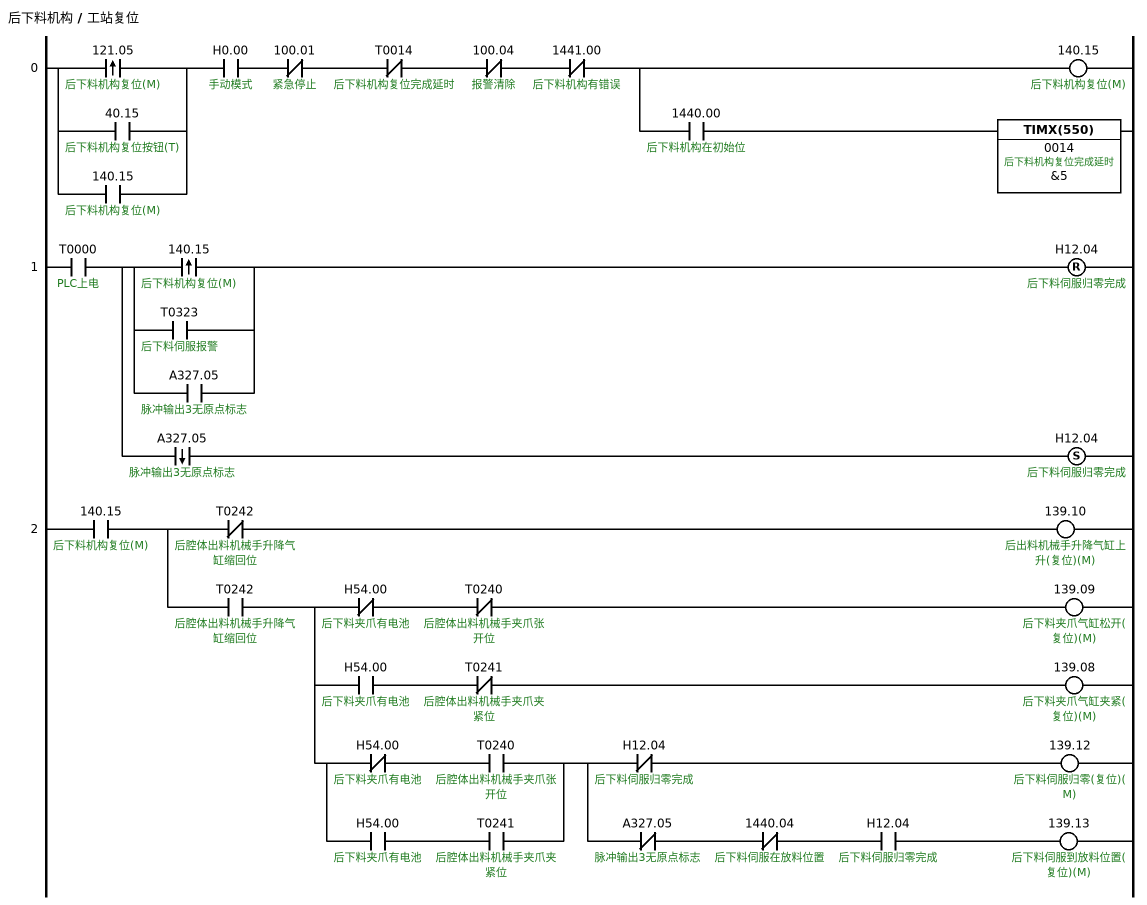
; [picture p216: 后下料机构 / 工站复位, rungs 0-2]
; rung 0
@LD 121.05  ; 后下料机构复位(M)
OR 40.15  ; 后下料机构复位按钮(T)
OR 140.15  ; 后下料机构复位(M)
AND H0.00  ; 手动模式
ANDNOT 100.01  ; 紧急停止
ANDNOT T0014  ; 后下料机构复位完成延时
ANDNOT 100.04  ; 报警清除
ANDNOT 1441.00  ; 后下料机构有错误
OUT 140.15  ; 后下料机构复位(M)
AND 1440.00  ; 后下料机构在初始位
TIMX(550) 0014 &5  ; 后下料机构复位完成延时
; rung 1
LD T0000  ; PLC上电
OUT TR0
@LD 140.15  ; 后下料机构复位(M)
OR T0323  ; 后下料伺服报警
OR A327.05  ; 脉冲输出3无原点标志
ANDLD
RSET H12.04  ; 后下料伺服归零完成
LD TR0
%AND A327.05  ; 脉冲输出3无原点标志
SET H12.04  ; 后下料伺服归零完成
; rung 2
LD 140.15  ; 后下料机构复位(M)
OUT TR0
ANDNOT T0242  ; 后腔体出料机械手升降气缸缩回位
OUT 139.10  ; 后出料机械手升降气缸上升(复位)(M)
LD TR0
AND T0242  ; 后腔体出料机械手升降气缸缩回位
OUT TR0
ANDNOT H54.00  ; 后下料夹爪有电池
ANDNOT T0240  ; 后腔体出料机械手夹爪张开位
OUT 139.09  ; 后下料夹爪气缸松开(复位)(M)
LD TR0
AND H54.00  ; 后下料夹爪有电池
ANDNOT T0241  ; 后腔体出料机械手夹爪夹紧位
OUT 139.08  ; 后下料夹爪气缸夹紧(复位)(M)
LD TR0
LDNOT H54.00  ; 后下料夹爪有电池
AND T0240  ; 后腔体出料机械手夹爪张开位
LD H54.00  ; 后下料夹爪有电池
AND T0241  ; 后腔体出料机械手夹爪夹紧位
ORLD
ANDLD
OUT TR0
ANDNOT H12.04  ; 后下料伺服归零完成
OUT 139.12  ; 后下料伺服归零(复位)(M)
LD TR0
ANDNOT A327.05  ; 脉冲输出3无原点标志
ANDNOT 1440.04  ; 后下料伺服在放料位置
AND H12.04  ; 后下料伺服归零完成
OUT 139.13  ; 后下料伺服到放料位置(复位)(M)

### Section 手动操作

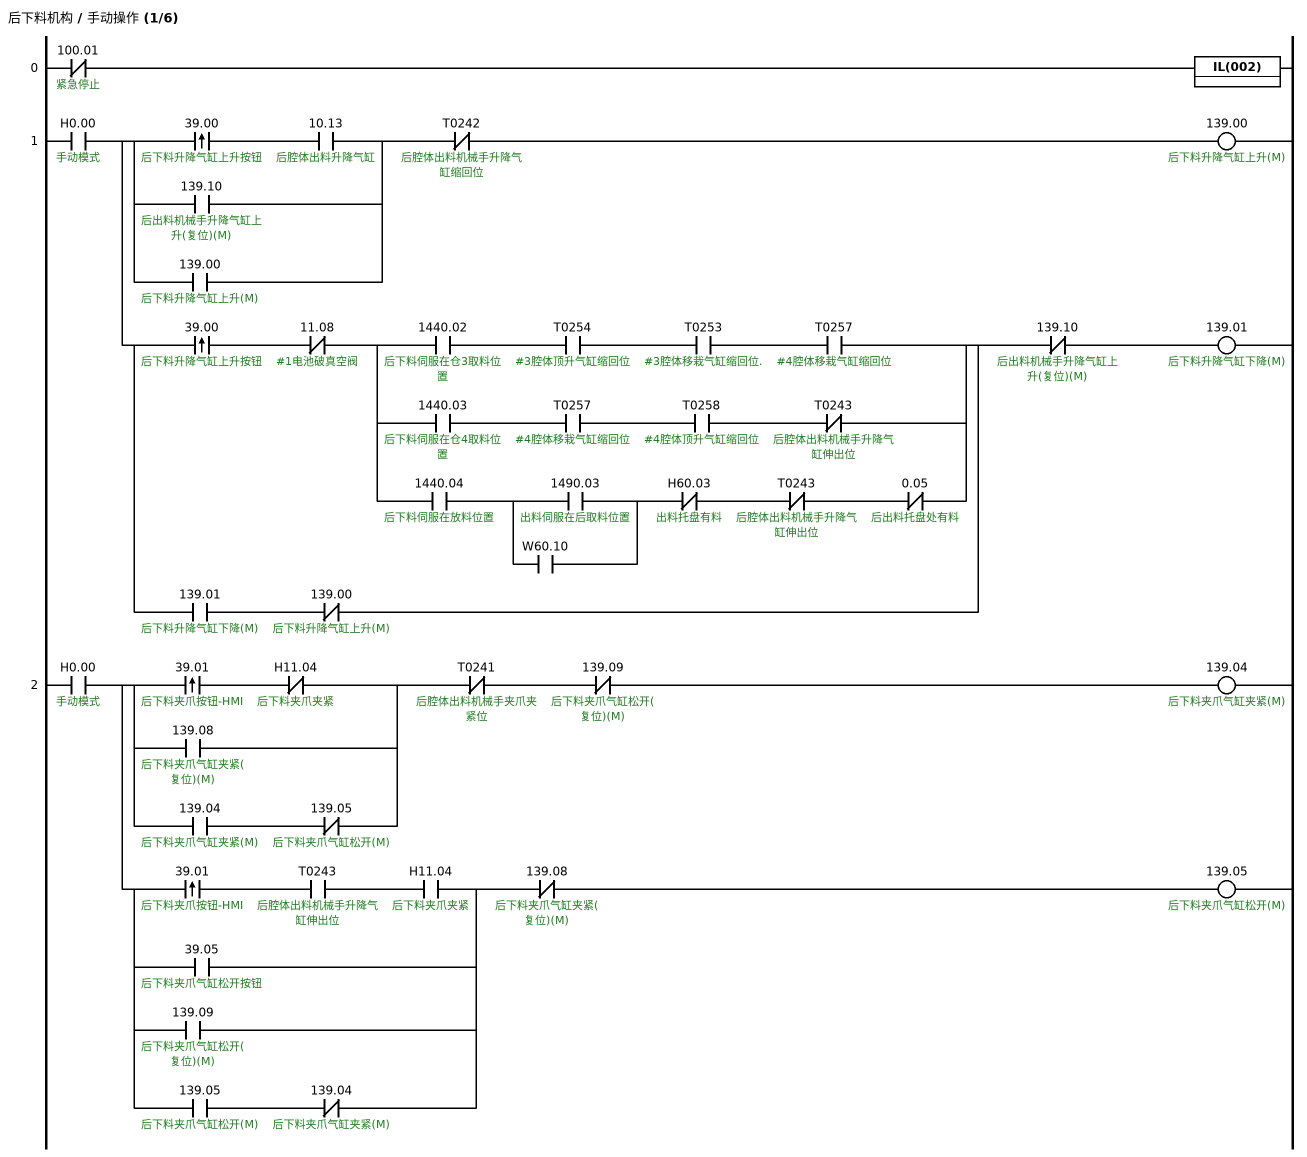
; rung 0
LDNOT 100.01  ; 紧急停止
IL(002)
; rung 1
LD H0.00  ; 手动模式
OUT TR0
@LD 39.00  ; 后下料升降气缸上升按钮
AND 10.13  ; 后腔体出料升降气缸
OR 139.10  ; 后出料机械手升降气缸上升(复位)(M)
OR 139.00  ; 后下料升降气缸上升(M)
ANDLD
ANDNOT T0242  ; 后腔体出料机械手升降气缸缩回位
OUT 139.00  ; 后下料升降气缸上升(M)
LD TR0
@LD 39.00  ; 后下料升降气缸上升按钮
ANDNOT 11.08  ; #1电池破真空阀
LD 1440.02  ; 后下料伺服在仓3取料位置
AND T0254  ; #3腔体顶升气缸缩回位
AND T0253  ; #3腔体移栽气缸缩回位.
AND T0257  ; #4腔体移栽气缸缩回位
LD 1440.03  ; 后下料伺服在仓4取料位置
AND T0257  ; #4腔体移栽气缸缩回位
AND T0258  ; #4腔体顶升气缸缩回位
ANDNOT T0243  ; 后腔体出料机械手升降气缸伸出位
ORLD
LD 1440.04  ; 后下料伺服在放料位置
LD 1490.03  ; 出料伺服在后取料位置
OR W60.10
ANDLD
ANDNOT H60.03  ; 出料托盘有料
ANDNOT T0243  ; 后腔体出料机械手升降气缸伸出位
ANDNOT 0.05  ; 后出料托盘处有料
ORLD
ANDLD
LD 139.01  ; 后下料升降气缸下降(M)
ANDNOT 139.00  ; 后下料升降气缸上升(M)
ORLD
ANDLD
ANDNOT 139.10  ; 后出料机械手升降气缸上升(复位)(M)
OUT 139.01  ; 后下料升降气缸下降(M)
; rung 2
LD H0.00  ; 手动模式
OUT TR0
@LD 39.01  ; 后下料夹爪按钮-HMI
ANDNOT H11.04  ; 后下料夹爪夹紧
OR 139.08  ; 后下料夹爪气缸夹紧(复位)(M)
LD 139.04  ; 后下料夹爪气缸夹紧(M)
ANDNOT 139.05  ; 后下料夹爪气缸松开(M)
ORLD
ANDLD
ANDNOT T0241  ; 后腔体出料机械手夹爪夹紧位
ANDNOT 139.09  ; 后下料夹爪气缸松开(复位)(M)
OUT 139.04  ; 后下料夹爪气缸夹紧(M)
LD TR0
@LD 39.01  ; 后下料夹爪按钮-HMI
AND T0243  ; 后腔体出料机械手升降气缸伸出位
AND H11.04  ; 后下料夹爪夹紧
OR 39.05  ; 后下料夹爪气缸松开按钮
OR 139.09  ; 后下料夹爪气缸松开(复位)(M)
LD 139.05  ; 后下料夹爪气缸松开(M)
ANDNOT 139.04  ; 后下料夹爪气缸夹紧(M)
ORLD
ANDLD
ANDNOT 139.08  ; 后下料夹爪气缸夹紧(复位)(M)
OUT 139.05  ; 后下料夹爪气缸松开(M)

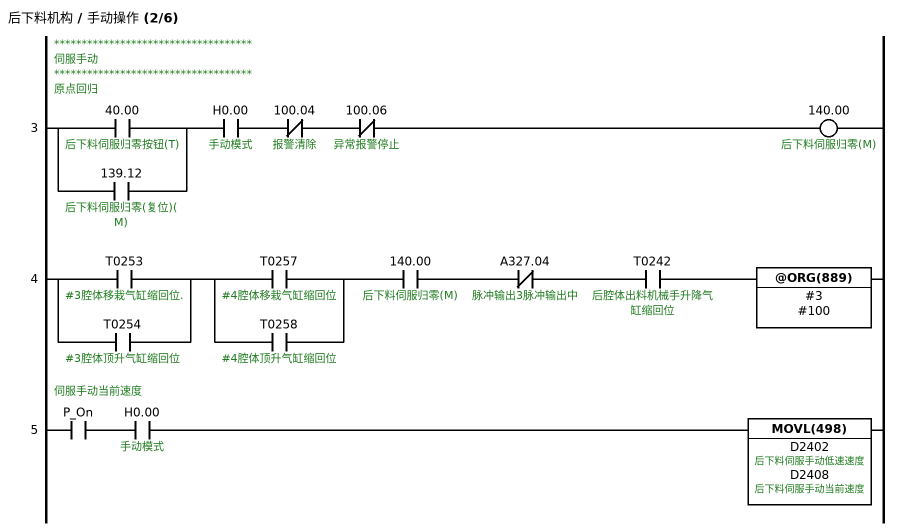
; rung 3: ************************************ / 伺服手动 / ************************************ / 原点回归
LD 40.00  ; 后下料伺服归零按钮(T)
OR 139.12  ; 后下料伺服归零(复位)(M)
AND H0.00  ; 手动模式
ANDNOT 100.04  ; 报警清除
ANDNOT 100.06  ; 异常报警停止
OUT 140.00  ; 后下料伺服归零(M)
; rung 4
LD T0253  ; #3腔体移栽气缸缩回位.
OR T0254  ; #3腔体顶升气缸缩回位
LD T0257  ; #4腔体移栽气缸缩回位
OR T0258  ; #4腔体顶升气缸缩回位
ANDLD
AND 140.00  ; 后下料伺服归零(M)
ANDNOT A327.04  ; 脉冲输出3脉冲输出中
AND T0242  ; 后腔体出料机械手升降气缸缩回位
@ORG(889) #3 #100
; rung 5: 伺服手动当前速度
LD P_On
AND H0.00  ; 手动模式
MOVL(498) D2402 D2408  ; 后下料伺服手动低速速度, 后下料伺服手动当前速度

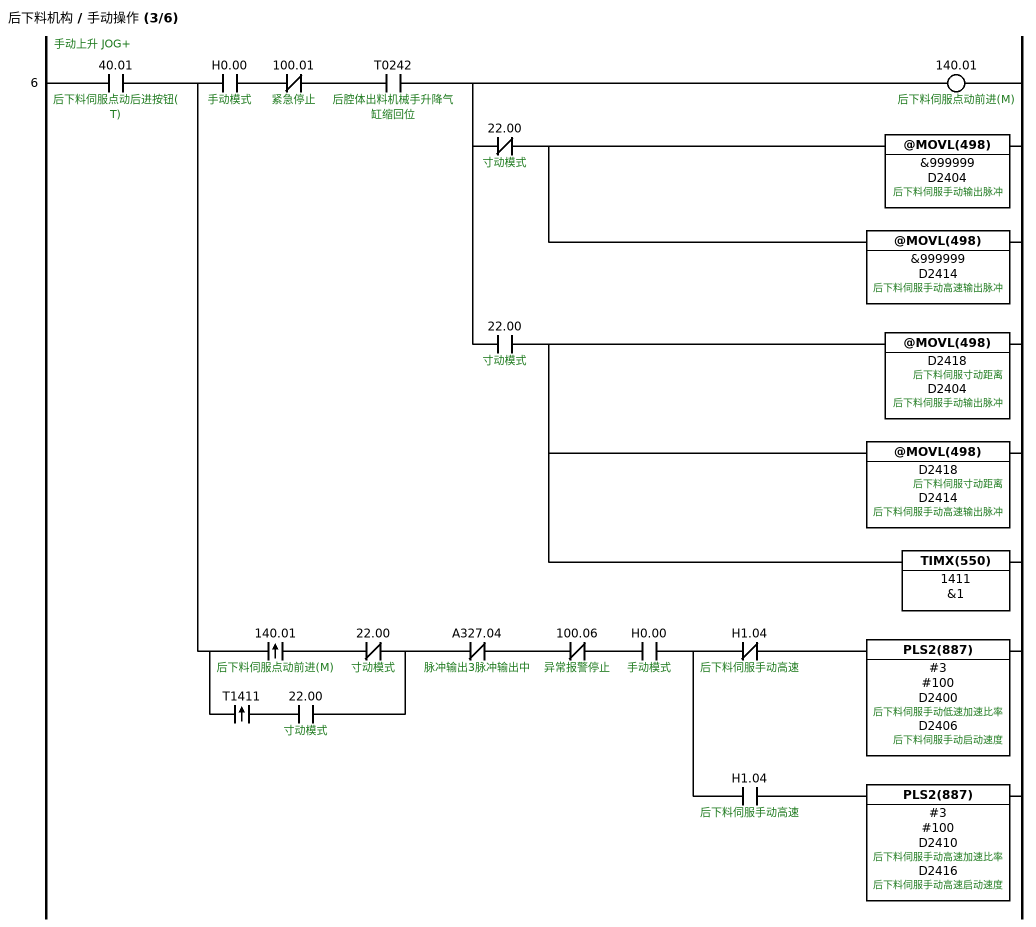
; rung 6: 手动上升 JOG+
LD 40.01  ; 后下料伺服点动后进按钮(T)
OUT TR0
AND H0.00  ; 手动模式
ANDNOT 100.01  ; 紧急停止
AND T0242  ; 后腔体出料机械手升降气缸缩回位
OUT TR1
OUT 140.01  ; 后下料伺服点动前进(M)
ANDNOT 22.00  ; 寸动模式
@MOVL(498) &999999 D2404  ; 后下料伺服手动输出脉冲
@MOVL(498) &999999 D2414  ; 后下料伺服手动高速输出脉冲
LD TR1
AND 22.00  ; 寸动模式
@MOVL(498) D2418 D2404  ; 后下料伺服寸动距离, 后下料伺服手动输出脉冲
@MOVL(498) D2418 D2414  ; 后下料伺服寸动距离, 后下料伺服手动高速输出脉冲
TIMX(550) 1411 &1
LD TR0
@LD 140.01  ; 后下料伺服点动前进(M)
ANDNOT 22.00  ; 寸动模式
@LD T1411
AND 22.00  ; 寸动模式
ORLD
ANDLD
ANDNOT A327.04  ; 脉冲输出3脉冲输出中
ANDNOT 100.06  ; 异常报警停止
AND H0.00  ; 手动模式
OUT TR0
ANDNOT H1.04  ; 后下料伺服手动高速
PLS2(887) #3 #100 D2400 D2406  ; 后下料伺服手动低速加速比率, 后下料伺服手动启动速度
LD TR0
AND H1.04  ; 后下料伺服手动高速
PLS2(887) #3 #100 D2410 D2416  ; 后下料伺服手动高速加速比率, 后下料伺服手动高速启动速度

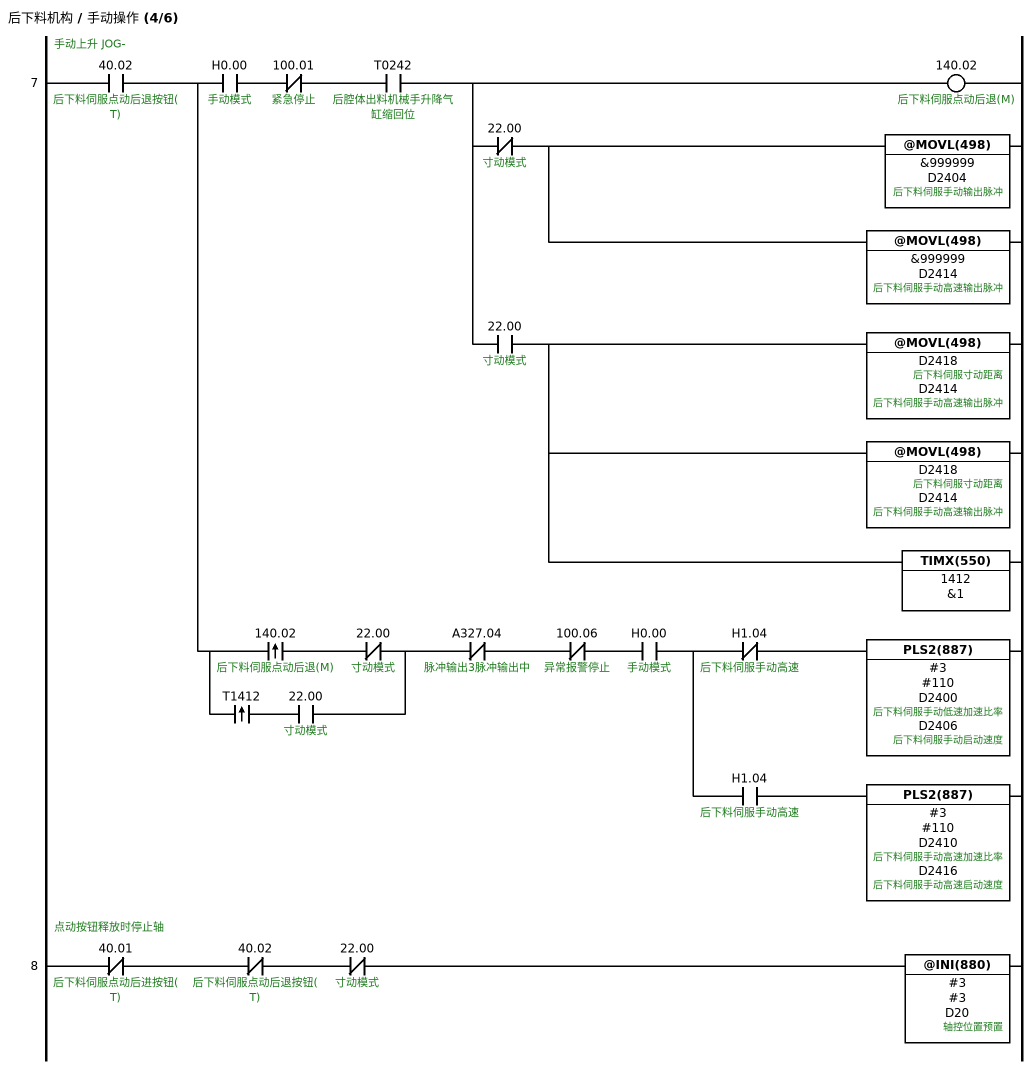
; rung 7: 手动上升 JOG-
LD 40.02  ; 后下料伺服点动后退按钮(T)
OUT TR0
AND H0.00  ; 手动模式
ANDNOT 100.01  ; 紧急停止
AND T0242  ; 后腔体出料机械手升降气缸缩回位
OUT TR1
OUT 140.02  ; 后下料伺服点动后退(M)
ANDNOT 22.00  ; 寸动模式
@MOVL(498) &999999 D2404  ; 后下料伺服手动输出脉冲
@MOVL(498) &999999 D2414  ; 后下料伺服手动高速输出脉冲
LD TR1
AND 22.00  ; 寸动模式
@MOVL(498) D2418 D2414  ; 后下料伺服寸动距离, 后下料伺服手动高速输出脉冲
@MOVL(498) D2418 D2414  ; 后下料伺服寸动距离, 后下料伺服手动高速输出脉冲
TIMX(550) 1412 &1
LD TR0
@LD 140.02  ; 后下料伺服点动后退(M)
ANDNOT 22.00  ; 寸动模式
@LD T1412
AND 22.00  ; 寸动模式
ORLD
ANDLD
ANDNOT A327.04  ; 脉冲输出3脉冲输出中
ANDNOT 100.06  ; 异常报警停止
AND H0.00  ; 手动模式
OUT TR0
ANDNOT H1.04  ; 后下料伺服手动高速
PLS2(887) #3 #110 D2400 D2406  ; 后下料伺服手动低速加速比率, 后下料伺服手动启动速度
LD TR0
AND H1.04  ; 后下料伺服手动高速
PLS2(887) #3 #110 D2410 D2416  ; 后下料伺服手动高速加速比率, 后下料伺服手动高速启动速度
; rung 8: 点动按钮释放时停止轴
LDNOT 40.01  ; 后下料伺服点动后进按钮(T)
ANDNOT 40.02  ; 后下料伺服点动后退按钮(T)
ANDNOT 22.00  ; 寸动模式
@INI(880) #3 #3 D20  ; 轴控位置预置

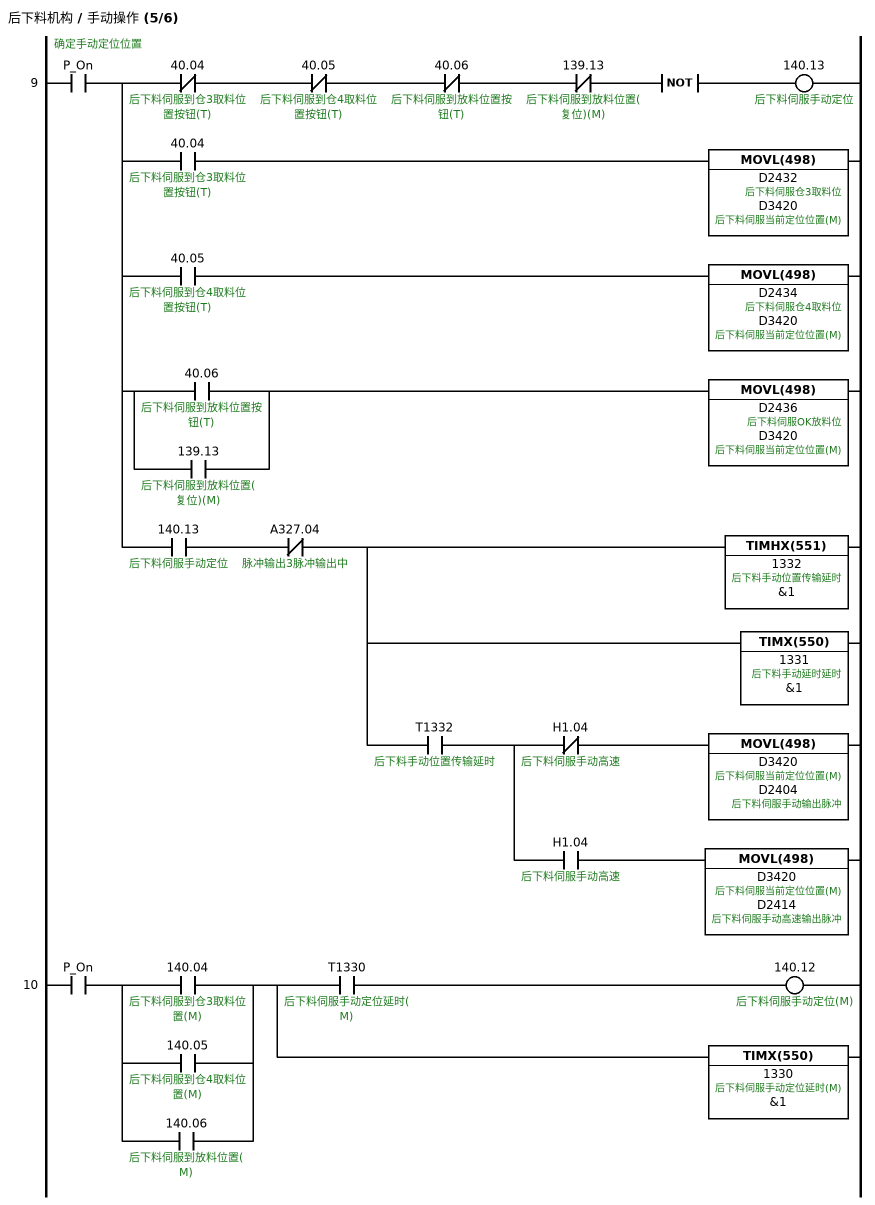
; rung 9: 确定手动定位位置
LD P_On
OUT TR0
ANDNOT 40.04  ; 后下料伺服到仓3取料位置按钮(T)
ANDNOT 40.05  ; 后下料伺服到仓4取料位置按钮(T)
ANDNOT 40.06  ; 后下料伺服到放料位置按钮(T)
ANDNOT 139.13  ; 后下料伺服到放料位置(复位)(M)
NOT(520)
OUT 140.13  ; 后下料伺服手动定位
LD TR0
AND 40.04  ; 后下料伺服到仓3取料位置按钮(T)
MOVL(498) D2432 D3420  ; 后下料伺服仓3取料位, 后下料伺服当前定位位置(M)
LD TR0
AND 40.05  ; 后下料伺服到仓4取料位置按钮(T)
MOVL(498) D2434 D3420  ; 后下料伺服仓4取料位, 后下料伺服当前定位位置(M)
LD TR0
LD 40.06  ; 后下料伺服到放料位置按钮(T)
OR 139.13  ; 后下料伺服到放料位置(复位)(M)
ANDLD
MOVL(498) D2436 D3420  ; 后下料伺服OK放料位, 后下料伺服当前定位位置(M)
LD TR0
AND 140.13  ; 后下料伺服手动定位
ANDNOT A327.04  ; 脉冲输出3脉冲输出中
TIMHX(551) 1332 &1  ; 后下料手动位置传输延时
TIMX(550) 1331 &1  ; 后下料手动延时延时
AND T1332  ; 后下料手动位置传输延时
OUT TR0
ANDNOT H1.04  ; 后下料伺服手动高速
MOVL(498) D3420 D2404  ; 后下料伺服当前定位位置(M), 后下料伺服手动输出脉冲
LD TR0
AND H1.04  ; 后下料伺服手动高速
MOVL(498) D3420 D2414  ; 后下料伺服当前定位位置(M), 后下料伺服手动高速输出脉冲
; rung 10
LD P_On
LD 140.04  ; 后下料伺服到仓3取料位置(M)
OR 140.05  ; 后下料伺服到仓4取料位置(M)
OR 140.06  ; 后下料伺服到放料位置(M)
ANDLD
OUT TR0
AND T1330  ; 后下料伺服手动定位延时(M)
OUT 140.12  ; 后下料伺服手动定位(M)
LD TR0
TIMX(550) 1330 &1  ; 后下料伺服手动定位延时(M)

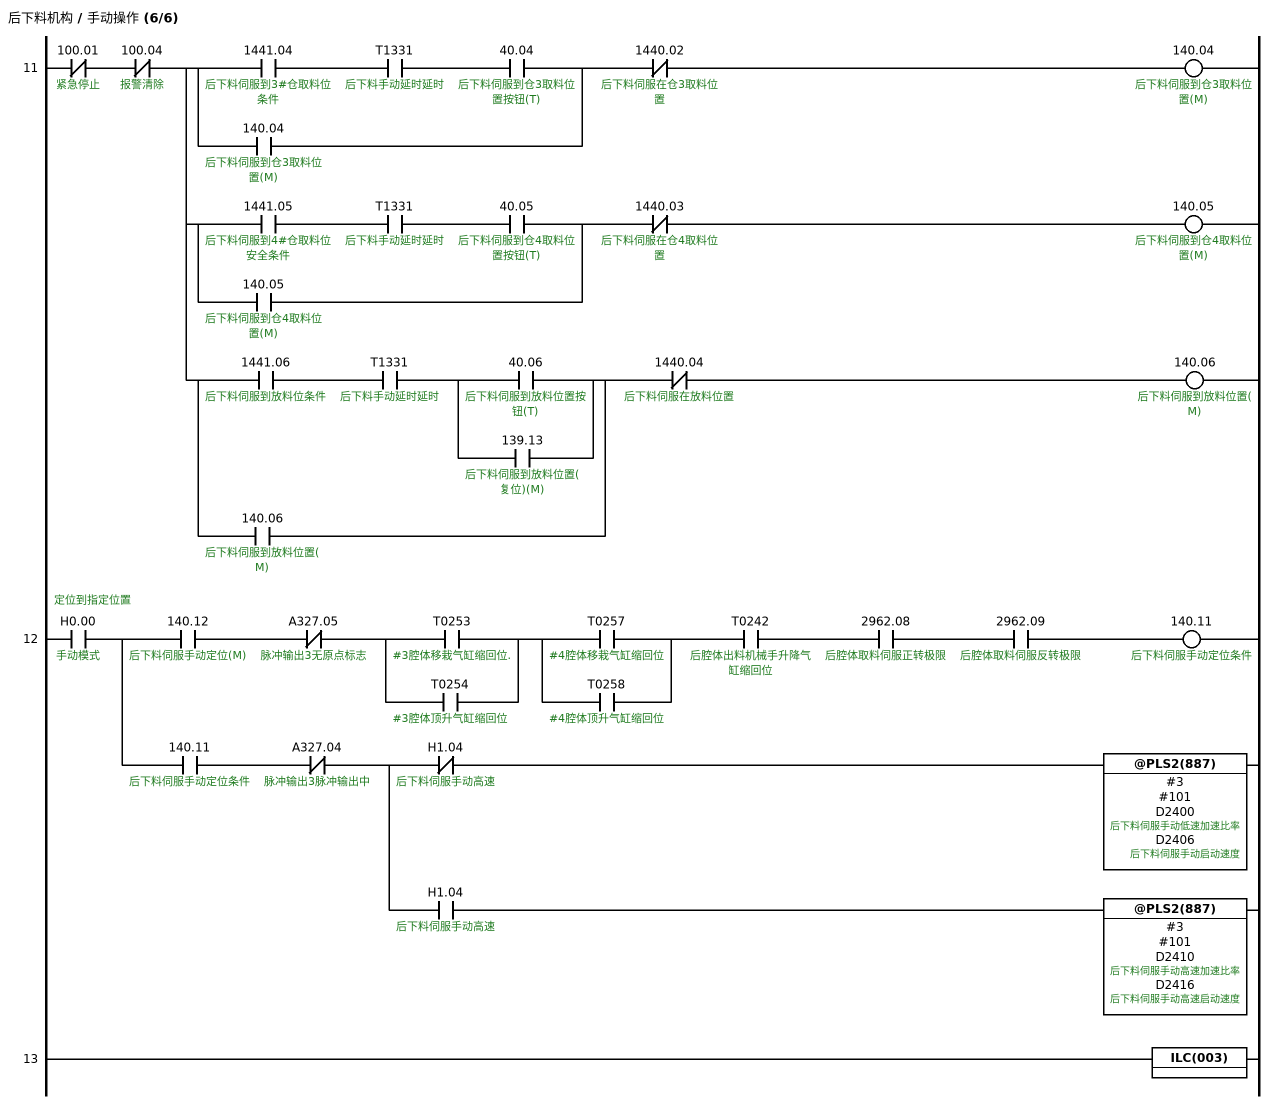
; rung 11
LDNOT 100.01  ; 紧急停止
ANDNOT 100.04  ; 报警清除
OUT TR0
LD 1441.04  ; 后下料伺服到3#仓取料位条件
AND T1331  ; 后下料手动延时延时
AND 40.04  ; 后下料伺服到仓3取料位置按钮(T)
OR 140.04  ; 后下料伺服到仓3取料位置(M)
ANDLD
ANDNOT 1440.02  ; 后下料伺服在仓3取料位置
OUT 140.04  ; 后下料伺服到仓3取料位置(M)
LD TR0
LD 1441.05  ; 后下料伺服到4#仓取料位安全条件
AND T1331  ; 后下料手动延时延时
AND 40.05  ; 后下料伺服到仓4取料位置按钮(T)
OR 140.05  ; 后下料伺服到仓4取料位置(M)
ANDLD
ANDNOT 1440.03  ; 后下料伺服在仓4取料位置
OUT 140.05  ; 后下料伺服到仓4取料位置(M)
LD TR0
LD 1441.06  ; 后下料伺服到放料位条件
AND T1331  ; 后下料手动延时延时
LD 40.06  ; 后下料伺服到放料位置按钮(T)
OR 139.13  ; 后下料伺服到放料位置(复位)(M)
ANDLD
OR 140.06  ; 后下料伺服到放料位置(M)
ANDLD
ANDNOT 1440.04  ; 后下料伺服在放料位置
OUT 140.06  ; 后下料伺服到放料位置(M)
; rung 12: 定位到指定位置
LD H0.00  ; 手动模式
OUT TR0
AND 140.12  ; 后下料伺服手动定位(M)
ANDNOT A327.05  ; 脉冲输出3无原点标志
LD T0253  ; #3腔体移栽气缸缩回位.
OR T0254  ; #3腔体顶升气缸缩回位
ANDLD
LD T0257  ; #4腔体移栽气缸缩回位
OR T0258  ; #4腔体顶升气缸缩回位
ANDLD
AND T0242  ; 后腔体出料机械手升降气缸缩回位
AND 2962.08  ; 后腔体取料伺服正转极限
AND 2962.09  ; 后腔体取料伺服反转极限
OUT 140.11  ; 后下料伺服手动定位条件
LD TR0
AND 140.11  ; 后下料伺服手动定位条件
ANDNOT A327.04  ; 脉冲输出3脉冲输出中
OUT TR0
ANDNOT H1.04  ; 后下料伺服手动高速
@PLS2(887) #3 #101 D2400 D2406  ; 后下料伺服手动低速加速比率, 后下料伺服手动启动速度
LD TR0
AND H1.04  ; 后下料伺服手动高速
@PLS2(887) #3 #101 D2410 D2416  ; 后下料伺服手动高速加速比率, 后下料伺服手动高速启动速度
; rung 13
ILC(003)

### Section 自动运行

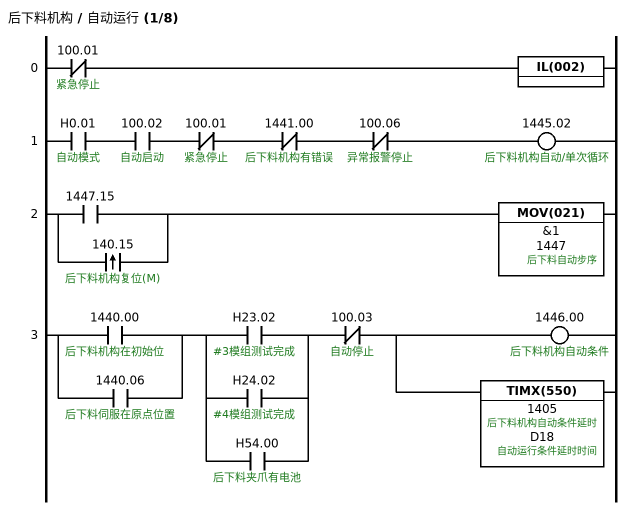
; rung 0
LDNOT 100.01  ; 紧急停止
IL(002)
; rung 1
LD H0.01  ; 自动模式
AND 100.02  ; 自动启动
ANDNOT 100.01  ; 紧急停止
ANDNOT 1441.00  ; 后下料机构有错误
ANDNOT 100.06  ; 异常报警停止
OUT 1445.02  ; 后下料机构自动/单次循环
; rung 2
LD 1447.15
@OR 140.15  ; 后下料机构复位(M)
MOV(021) &1 1447  ; 后下料自动步序
; rung 3
LD 1440.00  ; 后下料机构在初始位
OR 1440.06  ; 后下料伺服在原点位置
LD H23.02  ; #3模组测试完成
OR H24.02  ; #4模组测试完成
OR H54.00  ; 后下料夹爪有电池
ANDLD
ANDNOT 100.03  ; 自动停止
OUT 1446.00  ; 后下料机构自动条件
TIMX(550) 1405 D18  ; 自动运行条件延时时间, 后下料机构自动条件延时

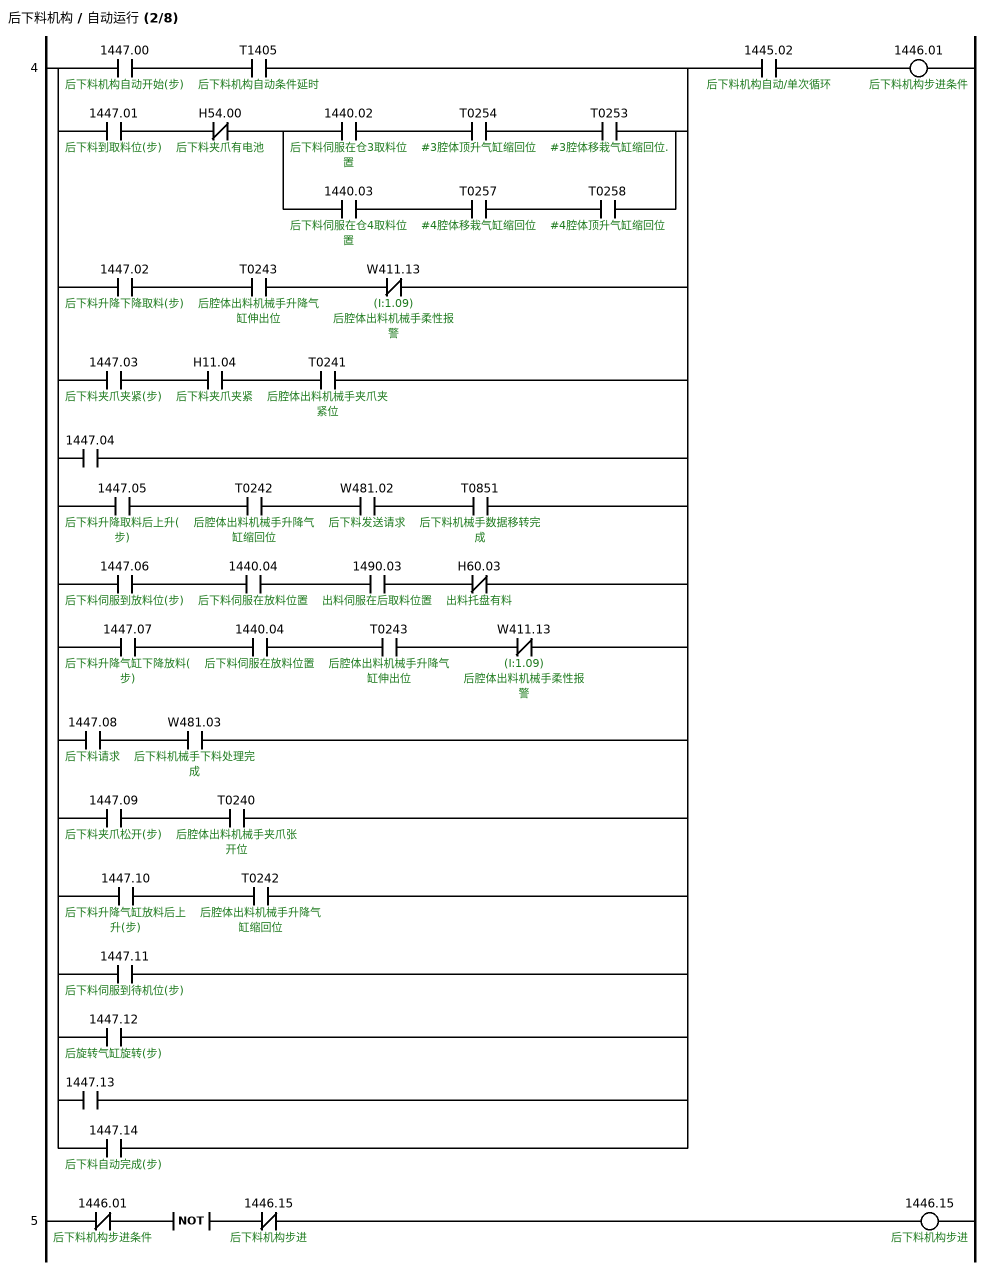
; rung 4
LD 1447.00  ; 后下料机构自动开始(步)
AND T1405  ; 后下料机构自动条件延时
LD 1447.01  ; 后下料到取料位(步)
ANDNOT H54.00  ; 后下料夹爪有电池
LD 1440.02  ; 后下料伺服在仓3取料位置
AND T0254  ; #3腔体顶升气缸缩回位
AND T0253  ; #3腔体移栽气缸缩回位.
LD 1440.03  ; 后下料伺服在仓4取料位置
AND T0257  ; #4腔体移栽气缸缩回位
AND T0258  ; #4腔体顶升气缸缩回位
ORLD
ANDLD
ORLD
LD 1447.02  ; 后下料升降下降取料(步)
AND T0243  ; 后腔体出料机械手升降气缸伸出位
ANDNOT W411.13  ; (I:1.09) 后腔体出料机械手柔性报警
ORLD
LD 1447.03  ; 后下料夹爪夹紧(步)
AND H11.04  ; 后下料夹爪夹紧
AND T0241  ; 后腔体出料机械手夹爪夹紧位
ORLD
OR 1447.04
LD 1447.05  ; 后下料升降取料后上升(步)
AND T0242  ; 后腔体出料机械手升降气缸缩回位
AND W481.02  ; 后下料发送请求
AND T0851  ; 后下料机械手数据移转完成
ORLD
LD 1447.06  ; 后下料伺服到放料位(步)
AND 1440.04  ; 后下料伺服在放料位置
AND 1490.03  ; 出料伺服在后取料位置
ANDNOT H60.03  ; 出料托盘有料
ORLD
LD 1447.07  ; 后下料升降气缸下降放料(步)
AND 1440.04  ; 后下料伺服在放料位置
AND T0243  ; 后腔体出料机械手升降气缸伸出位
ANDNOT W411.13  ; (I:1.09) 后腔体出料机械手柔性报警
ORLD
LD 1447.08  ; 后下料请求
AND W481.03  ; 后下料机械手下料处理完成
ORLD
LD 1447.09  ; 后下料夹爪松开(步)
AND T0240  ; 后腔体出料机械手夹爪张开位
ORLD
LD 1447.10  ; 后下料升降气缸放料后上升(步)
AND T0242  ; 后腔体出料机械手升降气缸缩回位
ORLD
OR 1447.11  ; 后下料伺服到待机位(步)
OR 1447.12  ; 后旋转气缸旋转(步)
OR 1447.13
OR 1447.14  ; 后下料自动完成(步)
AND 1445.02  ; 后下料机构自动/单次循环
OUT 1446.01  ; 后下料机构步进条件
; rung 5
LDNOT 1446.01  ; 后下料机构步进条件
NOT(520)
ANDNOT 1446.15  ; 后下料机构步进
OUT 1446.15  ; 后下料机构步进

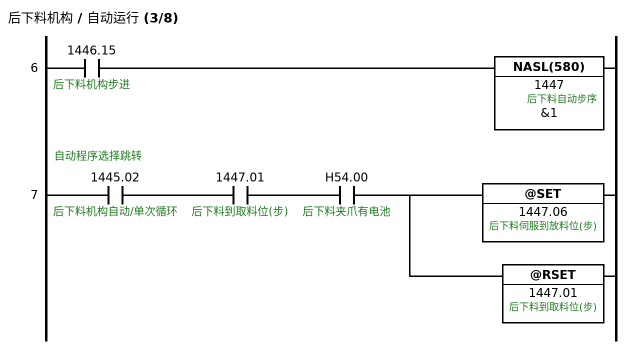
; rung 6
LD 1446.15  ; 后下料机构步进
NASL(580) 1447 &1  ; 后下料自动步序
; rung 7: 自动程序选择跳转
LD 1445.02  ; 后下料机构自动/单次循环
AND 1447.01  ; 后下料到取料位(步)
AND H54.00  ; 后下料夹爪有电池
@SET 1447.06  ; 后下料伺服到放料位(步)
@RSET 1447.01  ; 后下料到取料位(步)

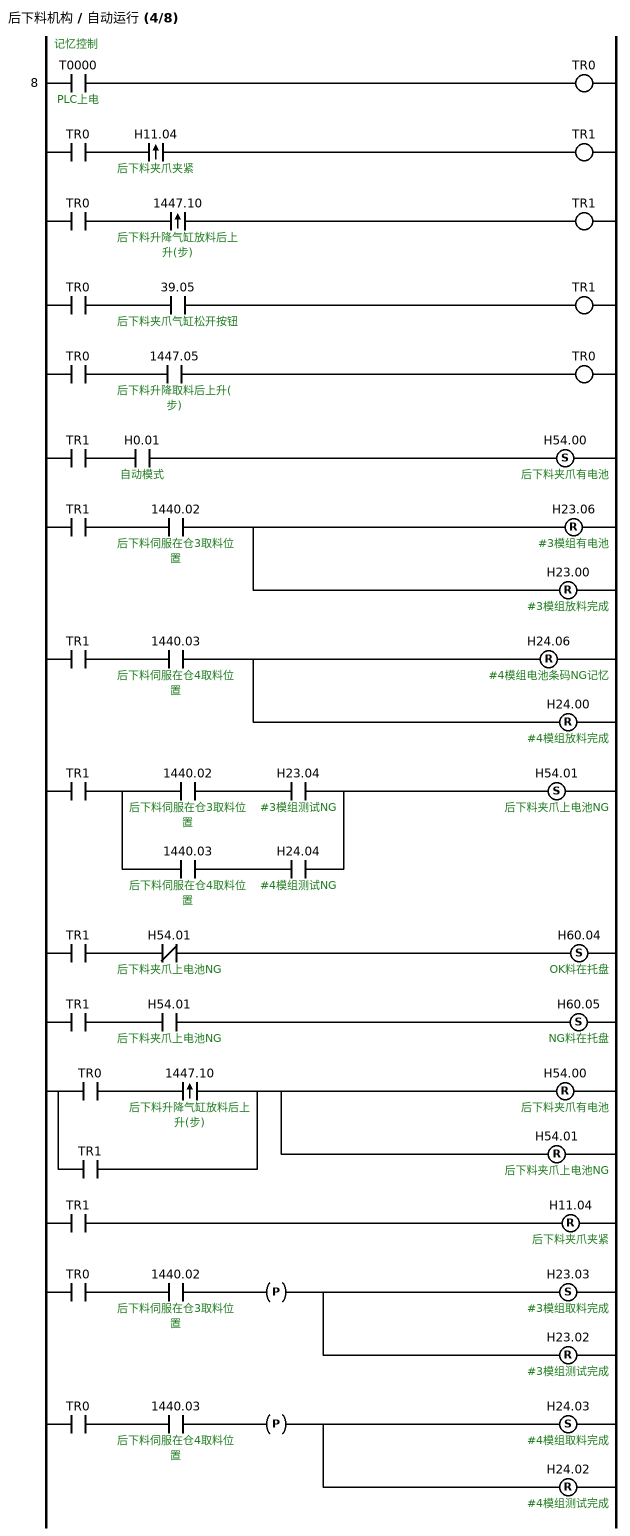
; rung 8: 记忆控制
LD T0000  ; PLC上电
OUT TR0
@AND H11.04  ; 后下料夹爪夹紧
OUT TR1
AND H0.01  ; 自动模式
SET H54.00  ; 后下料夹爪有电池
LD TR1
AND 1440.02  ; 后下料伺服在仓3取料位置
RSET H23.06  ; #3模组有电池
RSET H23.00  ; #3模组放料完成
LD TR1
AND 1440.03  ; 后下料伺服在仓4取料位置
RSET H24.06  ; #4模组电池条码NG记忆
RSET H24.00  ; #4模组放料完成
LD TR1
LD 1440.02  ; 后下料伺服在仓3取料位置
AND H23.04  ; #3模组测试NG
LD 1440.03  ; 后下料伺服在仓4取料位置
AND H24.04  ; #4模组测试NG
ORLD
ANDLD
SET H54.01  ; 后下料夹爪上电池NG
LD TR0
@AND 1447.10  ; 后下料升降气缸放料后上升(步)
OUT TR1
ANDNOT H54.01  ; 后下料夹爪上电池NG
SET H60.04  ; OK料在托盘
LD TR1
AND H54.01  ; 后下料夹爪上电池NG
SET H60.05  ; NG料在托盘
LD TR0
@AND 1447.10  ; 后下料升降气缸放料后上升(步)
LD TR0
AND 39.05  ; 后下料夹爪气缸松开按钮
OUT TR1
ORLD
RSET H54.00  ; 后下料夹爪有电池
RSET H54.01  ; 后下料夹爪上电池NG
LD TR1
RSET H11.04  ; 后下料夹爪夹紧
LD TR0
AND 1447.05  ; 后下料升降取料后上升(步)
OUT TR0
AND 1440.02  ; 后下料伺服在仓3取料位置
UP(521)
SET H23.03  ; #3模组取料完成
RSET H23.02  ; #3模组测试完成
LD TR0
AND 1440.03  ; 后下料伺服在仓4取料位置
UP(521)
SET H24.03  ; #4模组取料完成
RSET H24.02  ; #4模组测试完成

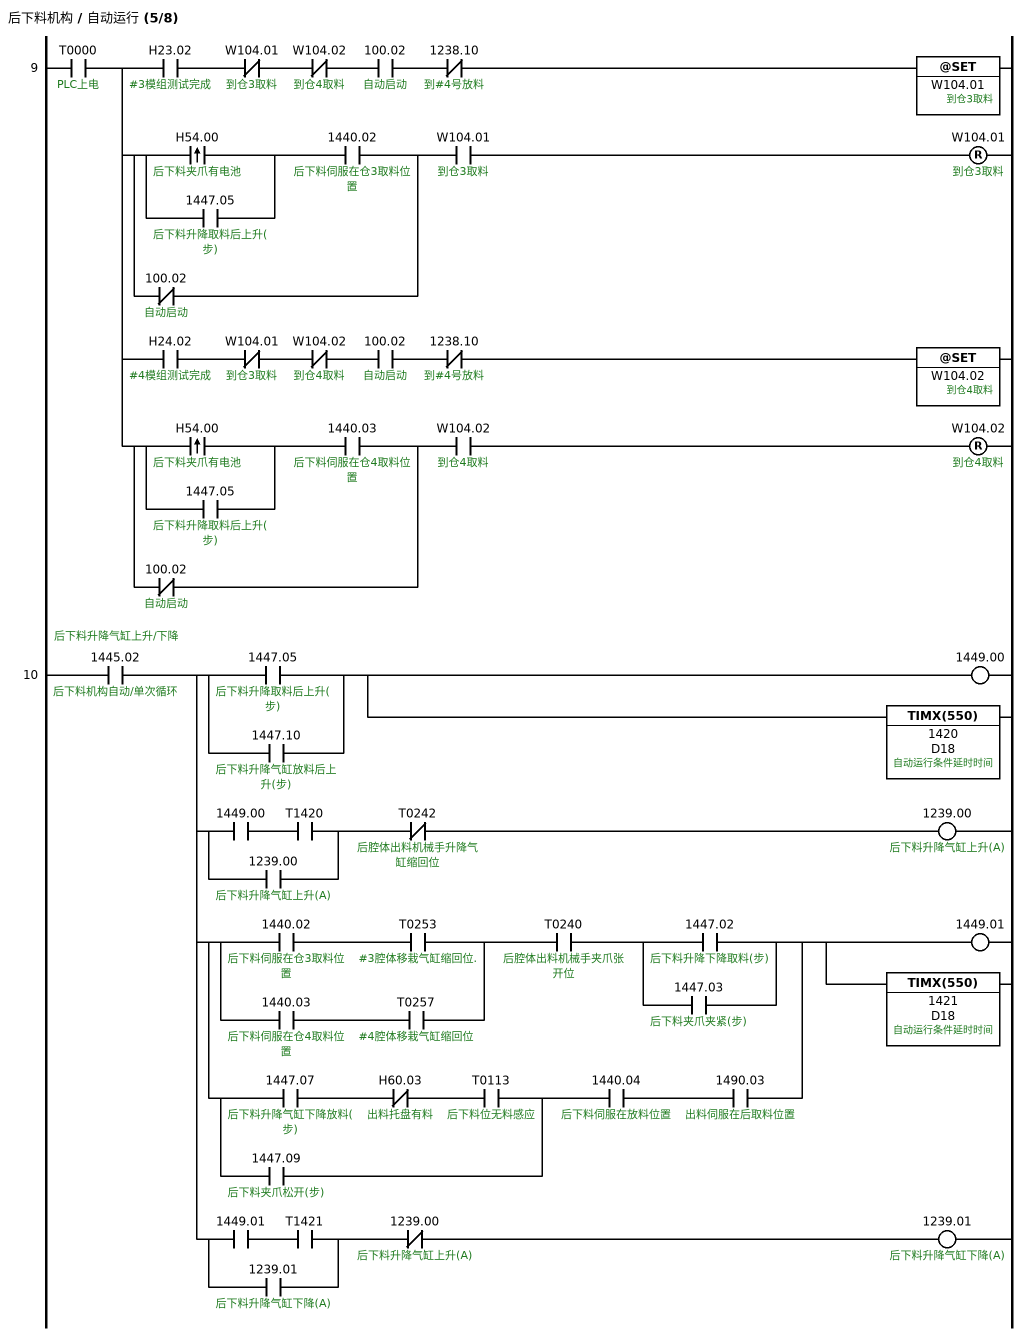
; rung 9
LD T0000  ; PLC上电
OUT TR0
AND H23.02  ; #3模组测试完成
ANDNOT W104.01  ; 到仓3取料
ANDNOT W104.02  ; 到仓4取料
AND 100.02  ; 自动启动
ANDNOT 1238.10  ; 到#4号放料
@SET W104.01  ; 到仓3取料
LD TR0
@LD H54.00  ; 后下料夹爪有电池
OR 1447.05  ; 后下料升降取料后上升(步)
AND 1440.02  ; 后下料伺服在仓3取料位置
ORNOT 100.02  ; 自动启动
ANDLD
AND W104.01  ; 到仓3取料
RSET W104.01  ; 到仓3取料
LD TR0
AND H24.02  ; #4模组测试完成
ANDNOT W104.01  ; 到仓3取料
ANDNOT W104.02  ; 到仓4取料
AND 100.02  ; 自动启动
ANDNOT 1238.10  ; 到#4号放料
@SET W104.02  ; 到仓4取料
LD TR0
@LD H54.00  ; 后下料夹爪有电池
OR 1447.05  ; 后下料升降取料后上升(步)
AND 1440.03  ; 后下料伺服在仓4取料位置
ORNOT 100.02  ; 自动启动
ANDLD
AND W104.02  ; 到仓4取料
RSET W104.02  ; 到仓4取料
; rung 10: 后下料升降气缸上升/下降
LD 1445.02  ; 后下料机构自动/单次循环
OUT TR0
LD 1447.05  ; 后下料升降取料后上升(步)
OR 1447.10  ; 后下料升降气缸放料后上升(步)
ANDLD
OUT 1449.00
TIMX(550) 1420 D18  ; 自动运行条件延时时间
LD TR0
LD 1449.00
AND T1420
OR 1239.00  ; 后下料升降气缸上升(A)
ANDLD
ANDNOT T0242  ; 后腔体出料机械手升降气缸缩回位
OUT 1239.00  ; 后下料升降气缸上升(A)
LD TR0
LD 1440.02  ; 后下料伺服在仓3取料位置
AND T0253  ; #3腔体移栽气缸缩回位.
LD 1440.03  ; 后下料伺服在仓4取料位置
AND T0257  ; #4腔体移栽气缸缩回位
ORLD
AND T0240  ; 后腔体出料机械手夹爪张开位
LD 1447.02  ; 后下料升降下降取料(步)
OR 1447.03  ; 后下料夹爪夹紧(步)
ANDLD
LD 1447.07  ; 后下料升降气缸下降放料(步)
ANDNOT H60.03  ; 出料托盘有料
AND T0113  ; 后下料位无料感应
OR 1447.09  ; 后下料夹爪松开(步)
AND 1440.04  ; 后下料伺服在放料位置
AND 1490.03  ; 出料伺服在后取料位置
ORLD
ANDLD
OUT 1449.01
TIMX(550) 1421 D18  ; 自动运行条件延时时间
LD TR0
LD 1449.01
AND T1421
OR 1239.01  ; 后下料升降气缸下降(A)
ANDLD
ANDNOT 1239.00  ; 后下料升降气缸上升(A)
OUT 1239.01  ; 后下料升降气缸下降(A)

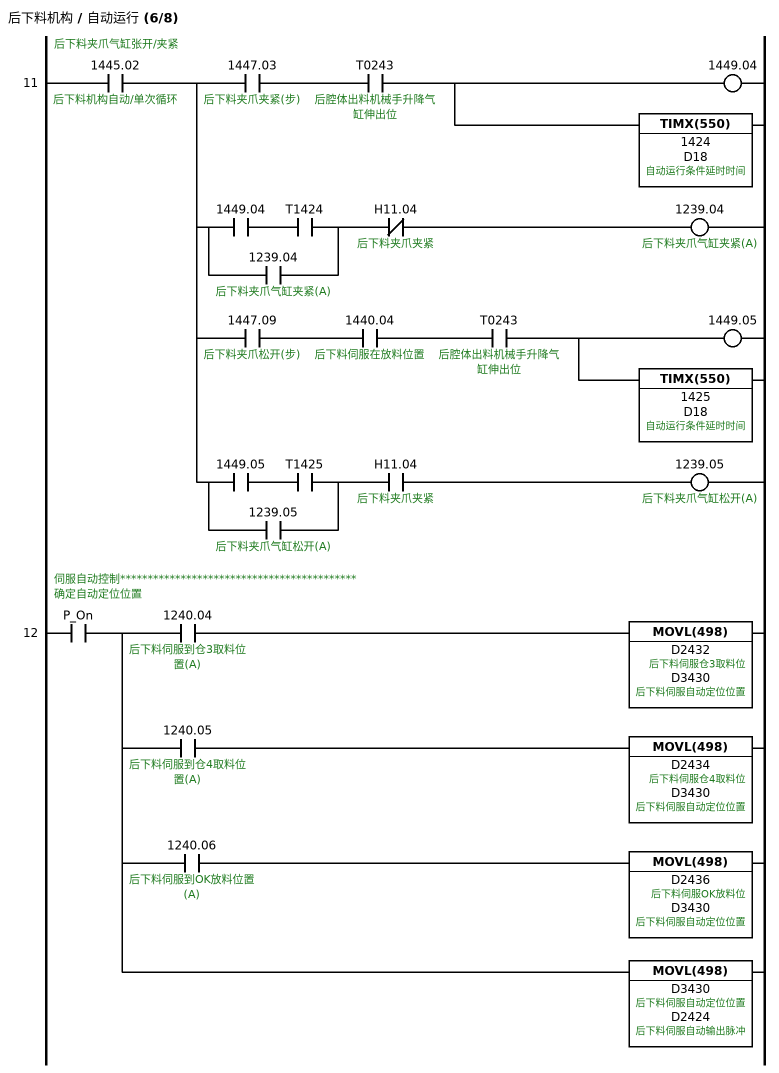
; rung 11: 后下料夹爪气缸张开/夹紧
LD 1445.02  ; 后下料机构自动/单次循环
OUT TR0
AND 1447.03  ; 后下料夹爪夹紧(步)
AND T0243  ; 后腔体出料机械手升降气缸伸出位
OUT 1449.04
TIMX(550) 1424 D18  ; 自动运行条件延时时间
LD TR0
LD 1449.04
AND T1424
OR 1239.04  ; 后下料夹爪气缸夹紧(A)
ANDLD
ANDNOT H11.04  ; 后下料夹爪夹紧
OUT 1239.04  ; 后下料夹爪气缸夹紧(A)
LD TR0
AND 1447.09  ; 后下料夹爪松开(步)
AND 1440.04  ; 后下料伺服在放料位置
AND T0243  ; 后腔体出料机械手升降气缸伸出位
OUT 1449.05
TIMX(550) 1425 D18  ; 自动运行条件延时时间
LD TR0
LD 1449.05
AND T1425
OR 1239.05  ; 后下料夹爪气缸松开(A)
ANDLD
AND H11.04  ; 后下料夹爪夹紧
OUT 1239.05  ; 后下料夹爪气缸松开(A)
; rung 12: 伺服自动控制******************************************* / 确定自动定位位置
LD P_On
OUT TR0
AND 1240.04  ; 后下料伺服到仓3取料位置(A)
MOVL(498) D2432 D3430  ; 后下料伺服仓3取料位, 后下料伺服自动定位位置
LD TR0
AND 1240.05  ; 后下料伺服到仓4取料位置(A)
MOVL(498) D2434 D3430  ; 后下料伺服仓4取料位, 后下料伺服自动定位位置
LD TR0
AND 1240.06  ; 后下料伺服到OK放料位置(A)
MOVL(498) D2436 D3430  ; 后下料伺服OK放料位, 后下料伺服自动定位位置
LD TR0
MOVL(498) D3430 D2424  ; 后下料伺服自动定位位置, 后下料伺服自动输出脉冲

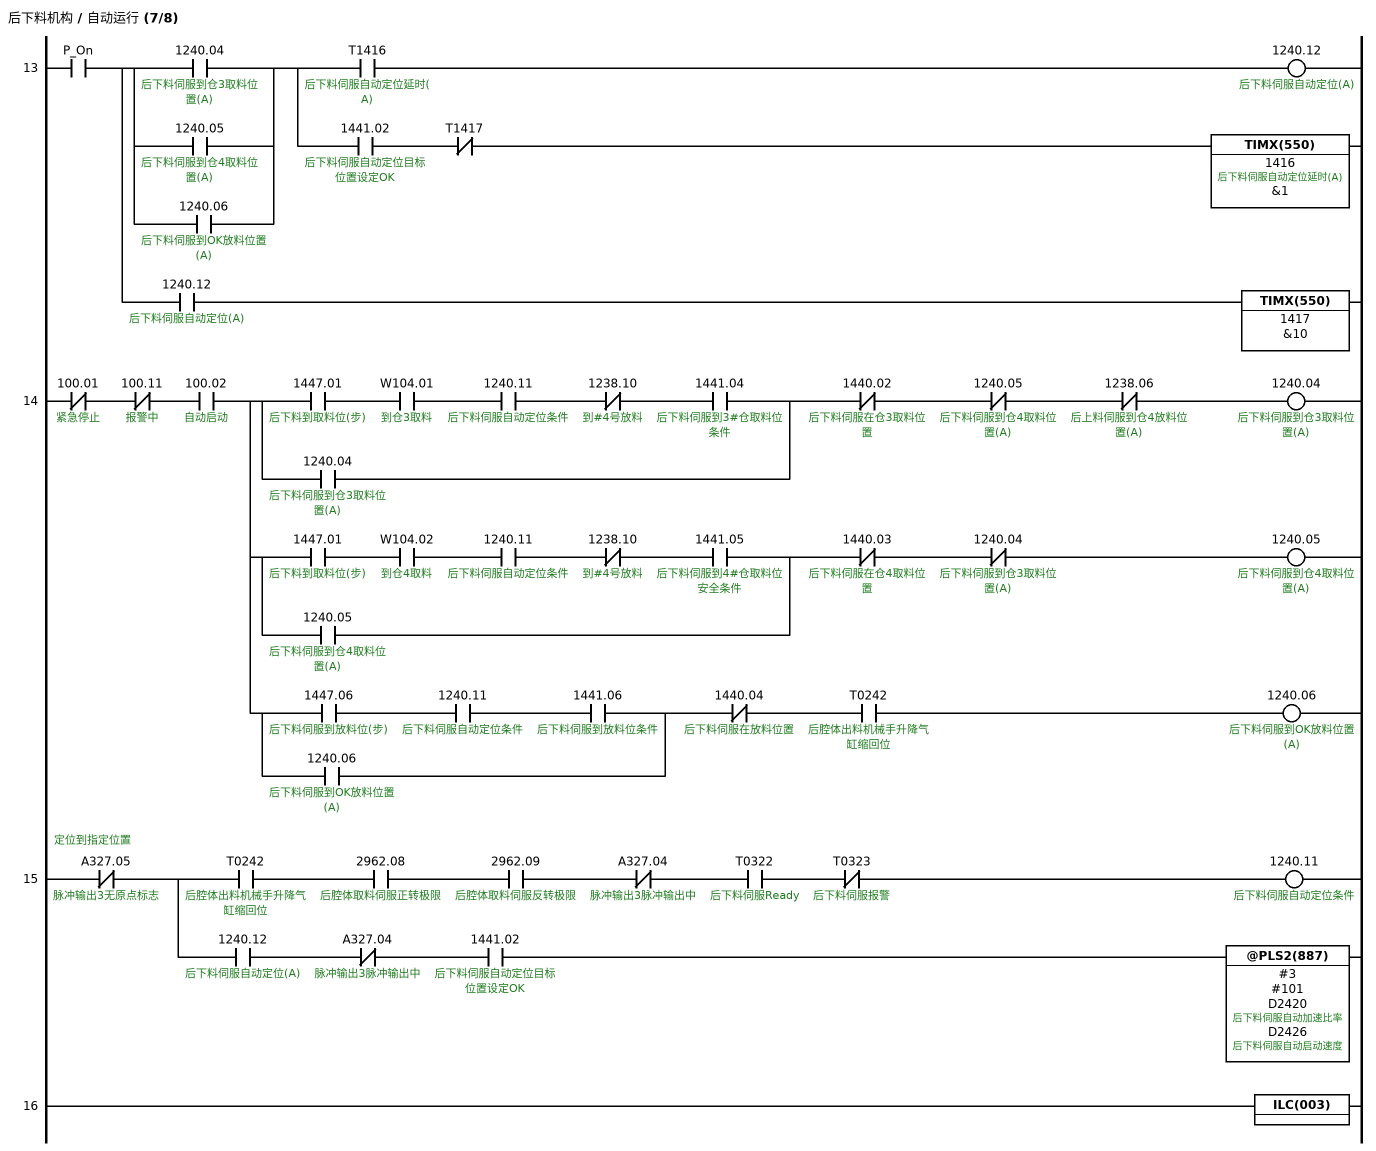
; rung 13
LD P_On
OUT TR0
LD 1240.04  ; 后下料伺服到仓3取料位置(A)
OR 1240.05  ; 后下料伺服到仓4取料位置(A)
OR 1240.06  ; 后下料伺服到OK放料位置(A)
ANDLD
OUT TR1
AND T1416  ; 后下料伺服自动定位延时(A)
OUT 1240.12  ; 后下料伺服自动定位(A)
LD TR1
AND 1441.02  ; 后下料伺服自动定位目标位置设定OK
ANDNOT T1417
TIMX(550) 1416 &1  ; 后下料伺服自动定位延时(A)
LD TR0
AND 1240.12  ; 后下料伺服自动定位(A)
TIMX(550) 1417 &10
; rung 14
LDNOT 100.01  ; 紧急停止
ANDNOT 100.11  ; 报警中
AND 100.02  ; 自动启动
OUT TR0
LD 1447.01  ; 后下料到取料位(步)
AND W104.01  ; 到仓3取料
AND 1240.11  ; 后下料伺服自动定位条件
ANDNOT 1238.10  ; 到#4号放料
AND 1441.04  ; 后下料伺服到3#仓取料位条件
OR 1240.04  ; 后下料伺服到仓3取料位置(A)
ANDLD
ANDNOT 1440.02  ; 后下料伺服在仓3取料位置
ANDNOT 1240.05  ; 后下料伺服到仓4取料位置(A)
ANDNOT 1238.06  ; 后上料伺服到仓4放料位置(A)
OUT 1240.04  ; 后下料伺服到仓3取料位置(A)
LD TR0
LD 1447.01  ; 后下料到取料位(步)
AND W104.02  ; 到仓4取料
AND 1240.11  ; 后下料伺服自动定位条件
ANDNOT 1238.10  ; 到#4号放料
AND 1441.05  ; 后下料伺服到4#仓取料位安全条件
OR 1240.05  ; 后下料伺服到仓4取料位置(A)
ANDLD
ANDNOT 1440.03  ; 后下料伺服在仓4取料位置
ANDNOT 1240.04  ; 后下料伺服到仓3取料位置(A)
OUT 1240.05  ; 后下料伺服到仓4取料位置(A)
LD TR0
LD 1447.06  ; 后下料伺服到放料位(步)
AND 1240.11  ; 后下料伺服自动定位条件
AND 1441.06  ; 后下料伺服到放料位条件
OR 1240.06  ; 后下料伺服到OK放料位置(A)
ANDLD
ANDNOT 1440.04  ; 后下料伺服在放料位置
AND T0242  ; 后腔体出料机械手升降气缸缩回位
OUT 1240.06  ; 后下料伺服到OK放料位置(A)
; rung 15: 定位到指定位置
LDNOT A327.05  ; 脉冲输出3无原点标志
OUT TR0
AND T0242  ; 后腔体出料机械手升降气缸缩回位
AND 2962.08  ; 后腔体取料伺服正转极限
AND 2962.09  ; 后腔体取料伺服反转极限
ANDNOT A327.04  ; 脉冲输出3脉冲输出中
AND T0322  ; 后下料伺服Ready
ANDNOT T0323  ; 后下料伺服报警
OUT 1240.11  ; 后下料伺服自动定位条件
LD TR0
AND 1240.12  ; 后下料伺服自动定位(A)
ANDNOT A327.04  ; 脉冲输出3脉冲输出中
AND 1441.02  ; 后下料伺服自动定位目标位置设定OK
@PLS2(887) #3 #101 D2420 D2426  ; 后下料伺服自动加速比率, 后下料伺服自动启动速度
; rung 16
ILC(003)

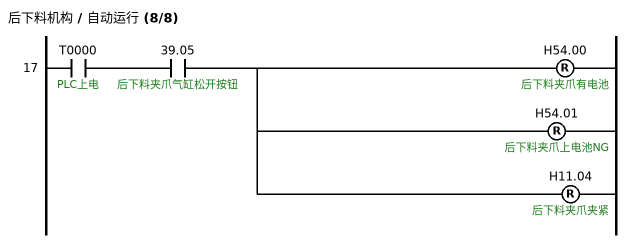
; rung 17
LD T0000  ; PLC上电
AND 39.05  ; 后下料夹爪气缸松开按钮
RSET H54.00  ; 后下料夹爪有电池
RSET H54.01  ; 后下料夹爪上电池NG
RSET H11.04  ; 后下料夹爪夹紧

### Section 外部输出

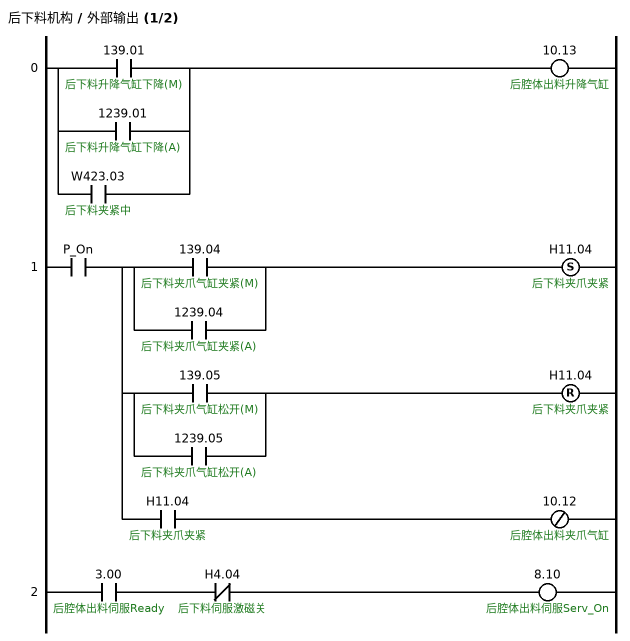
; rung 0
LD 139.01  ; 后下料升降气缸下降(M)
OR 1239.01  ; 后下料升降气缸下降(A)
OR W423.03  ; 后下料夹紧中
OUT 10.13  ; 后腔体出料升降气缸
; rung 1
LD P_On
OUT TR0
LD 139.04  ; 后下料夹爪气缸夹紧(M)
OR 1239.04  ; 后下料夹爪气缸夹紧(A)
ANDLD
SET H11.04  ; 后下料夹爪夹紧
LD TR0
LD 139.05  ; 后下料夹爪气缸松开(M)
OR 1239.05  ; 后下料夹爪气缸松开(A)
ANDLD
RSET H11.04  ; 后下料夹爪夹紧
LD TR0
AND H11.04  ; 后下料夹爪夹紧
OUTNOT 10.12  ; 后腔体出料夹爪气缸
; rung 2
LD 3.00  ; 后腔体出料伺服Ready
ANDNOT H4.04  ; 后下料伺服激磁关
OUT 8.10  ; 后腔体出料伺服Serv_On

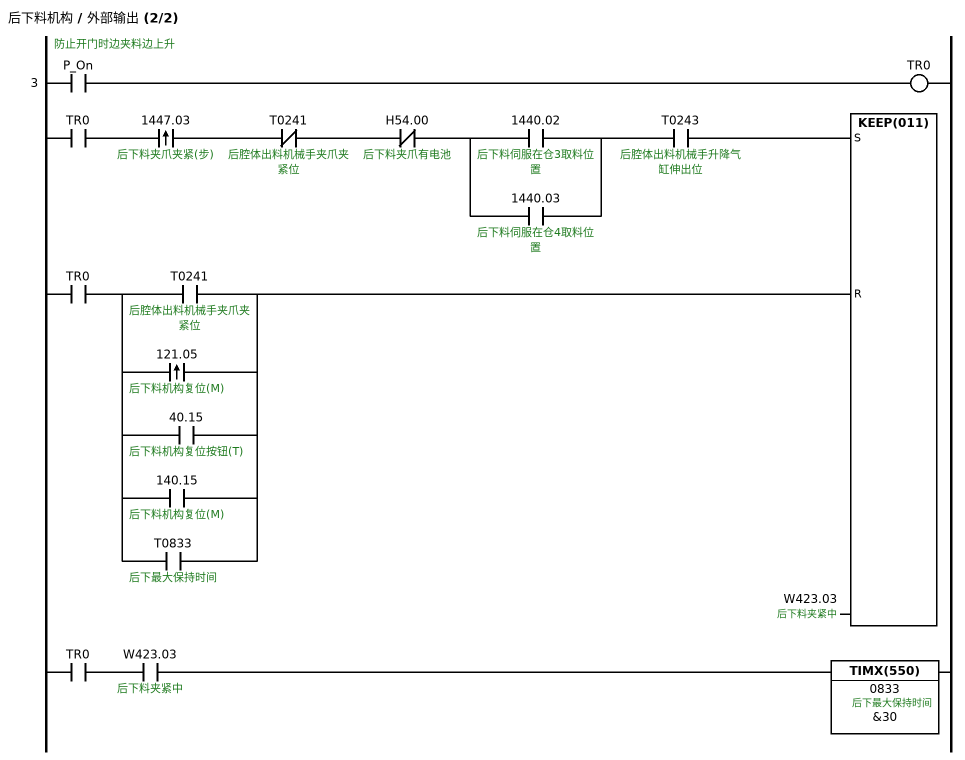
; rung 3: 防止开门时边夹料边上升
LD P_On
OUT TR0
@AND 1447.03  ; 后下料夹爪夹紧(步)
ANDNOT T0241  ; 后腔体出料机械手夹爪夹紧位
ANDNOT H54.00  ; 后下料夹爪有电池
LD 1440.02  ; 后下料伺服在仓3取料位置
OR 1440.03  ; 后下料伺服在仓4取料位置
ANDLD
AND T0243  ; 后腔体出料机械手升降气缸伸出位
LD TR0
LD T0241  ; 后腔体出料机械手夹爪夹紧位
@OR 121.05  ; 后下料机构复位(M)
OR 40.15  ; 后下料机构复位按钮(T)
OR 140.15  ; 后下料机构复位(M)
OR T0833  ; 后下最大保持时间
ANDLD
KEEP(011) W423.03  ; 后下料夹紧中
LD TR0
AND W423.03  ; 后下料夹紧中
TIMX(550) 0833 &30  ; 后下最大保持时间

### Section 指示灯
; rung 0: ************************************************** / 气缸动作及位置指示灯

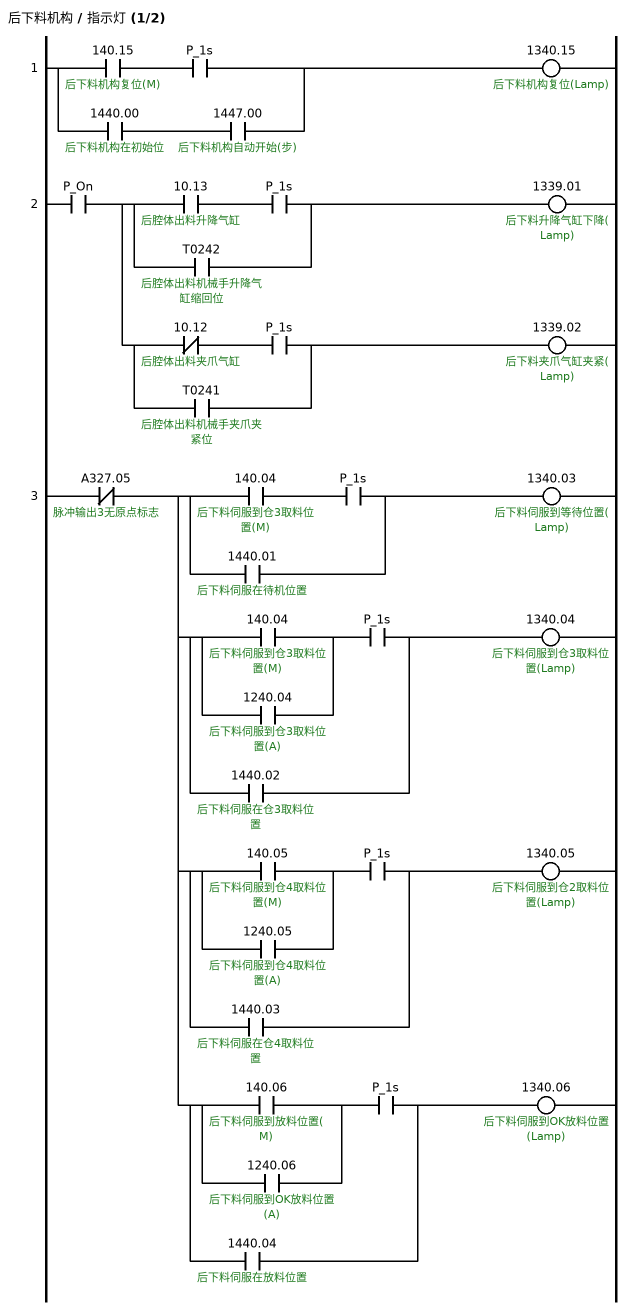
; rung 1
LD 140.15  ; 后下料机构复位(M)
AND P_1s
LD 1440.00  ; 后下料机构在初始位
AND 1447.00  ; 后下料机构自动开始(步)
ORLD
OUT 1340.15  ; 后下料机构复位(Lamp)
; rung 2
LD P_On
OUT TR0
LD 10.13  ; 后腔体出料升降气缸
AND P_1s
OR T0242  ; 后腔体出料机械手升降气缸缩回位
ANDLD
OUT 1339.01  ; 后下料升降气缸下降(Lamp)
LD TR0
LDNOT 10.12  ; 后腔体出料夹爪气缸
AND P_1s
OR T0241  ; 后腔体出料机械手夹爪夹紧位
ANDLD
OUT 1339.02  ; 后下料夹爪气缸夹紧(Lamp)
; rung 3
LDNOT A327.05  ; 脉冲输出3无原点标志
OUT TR0
LD 140.04  ; 后下料伺服到仓3取料位置(M)
AND P_1s
OR 1440.01  ; 后下料伺服在待机位置
ANDLD
OUT 1340.03  ; 后下料伺服到等待位置(Lamp)
LD TR0
LD 140.04  ; 后下料伺服到仓3取料位置(M)
OR 1240.04  ; 后下料伺服到仓3取料位置(A)
AND P_1s
OR 1440.02  ; 后下料伺服在仓3取料位置
ANDLD
OUT 1340.04  ; 后下料伺服到仓3取料位置(Lamp)
LD TR0
LD 140.05  ; 后下料伺服到仓4取料位置(M)
OR 1240.05  ; 后下料伺服到仓4取料位置(A)
AND P_1s
OR 1440.03  ; 后下料伺服在仓4取料位置
ANDLD
OUT 1340.05  ; 后下料伺服到仓2取料位置(Lamp)
LD TR0
LD 140.06  ; 后下料伺服到放料位置(M)
OR 1240.06  ; 后下料伺服到OK放料位置(A)
AND P_1s
OR 1440.04  ; 后下料伺服在放料位置
ANDLD
OUT 1340.06  ; 后下料伺服到OK放料位置(Lamp)

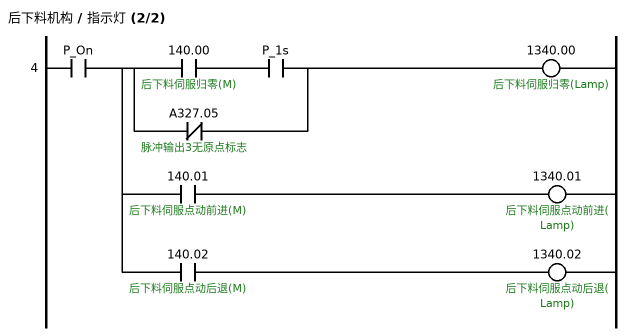
; rung 4
LD P_On
OUT TR0
LD 140.00  ; 后下料伺服归零(M)
AND P_1s
ORNOT A327.05  ; 脉冲输出3无原点标志
ANDLD
OUT 1340.00  ; 后下料伺服归零(Lamp)
LD TR0
AND 140.01  ; 后下料伺服点动前进(M)
OUT 1340.01  ; 后下料伺服点动前进(Lamp)
LD TR0
AND 140.02  ; 后下料伺服点动后退(M)
OUT 1340.02  ; 后下料伺服点动后退(Lamp)

### Section END
; rung 0
END(001)

## Program 腔体机构 (cyclic task 6)

### Section Main

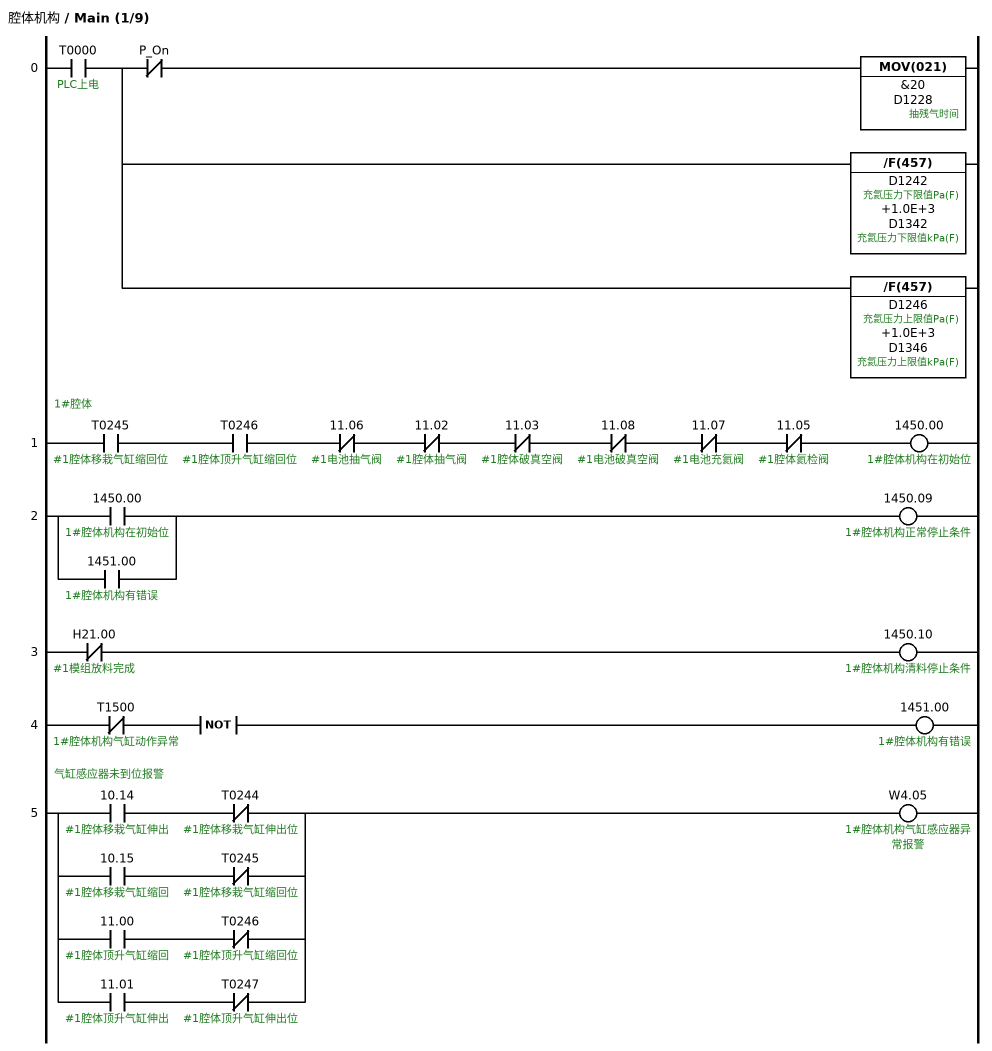
; rung 0
LD T0000  ; PLC上电
OUT TR0
ANDNOT P_On
MOV(021) &20 D1228  ; 抽残气时间
LD TR0
/F(457) D1242 +1.0E+3 D1342  ; 充氦压力下限值Pa(F), 充氦压力下限值kPa(F)
/F(457) D1246 +1.0E+3 D1346  ; 充氦压力上限值Pa(F), 充氦压力上限值kPa(F)
; rung 1: 1#腔体
LD T0245  ; #1腔体移栽气缸缩回位
AND T0246  ; #1腔体顶升气缸缩回位
ANDNOT 11.06  ; #1电池抽气阀
ANDNOT 11.02  ; #1腔体抽气阀
ANDNOT 11.03  ; #1腔体破真空阀
ANDNOT 11.08  ; #1电池破真空阀
ANDNOT 11.07  ; #1电池充氦阀
ANDNOT 11.05  ; #1腔体氦检阀
OUT 1450.00  ; 1#腔体机构在初始位
; rung 2
LD 1450.00  ; 1#腔体机构在初始位
OR 1451.00  ; 1#腔体机构有错误
OUT 1450.09  ; 1#腔体机构正常停止条件
; rung 3
LDNOT H21.00  ; #1模组放料完成
OUT 1450.10  ; 1#腔体机构清料停止条件
; rung 4
LDNOT T1500  ; 1#腔体机构气缸动作异常
NOT(520)
OUT 1451.00  ; 1#腔体机构有错误
; rung 5: 气缸感应器未到位报警
LD 10.14  ; #1腔体移栽气缸伸出
ANDNOT T0244  ; #1腔体移栽气缸伸出位
LD 10.15  ; #1腔体移栽气缸缩回
ANDNOT T0245  ; #1腔体移栽气缸缩回位
ORLD
LD 11.00  ; #1腔体顶升气缸缩回
ANDNOT T0246  ; #1腔体顶升气缸缩回位
ORLD
LD 11.01  ; #1腔体顶升气缸伸出
ANDNOT T0247  ; #1腔体顶升气缸伸出位
ORLD
OUT W4.05  ; 1#腔体机构气缸感应器异常报警

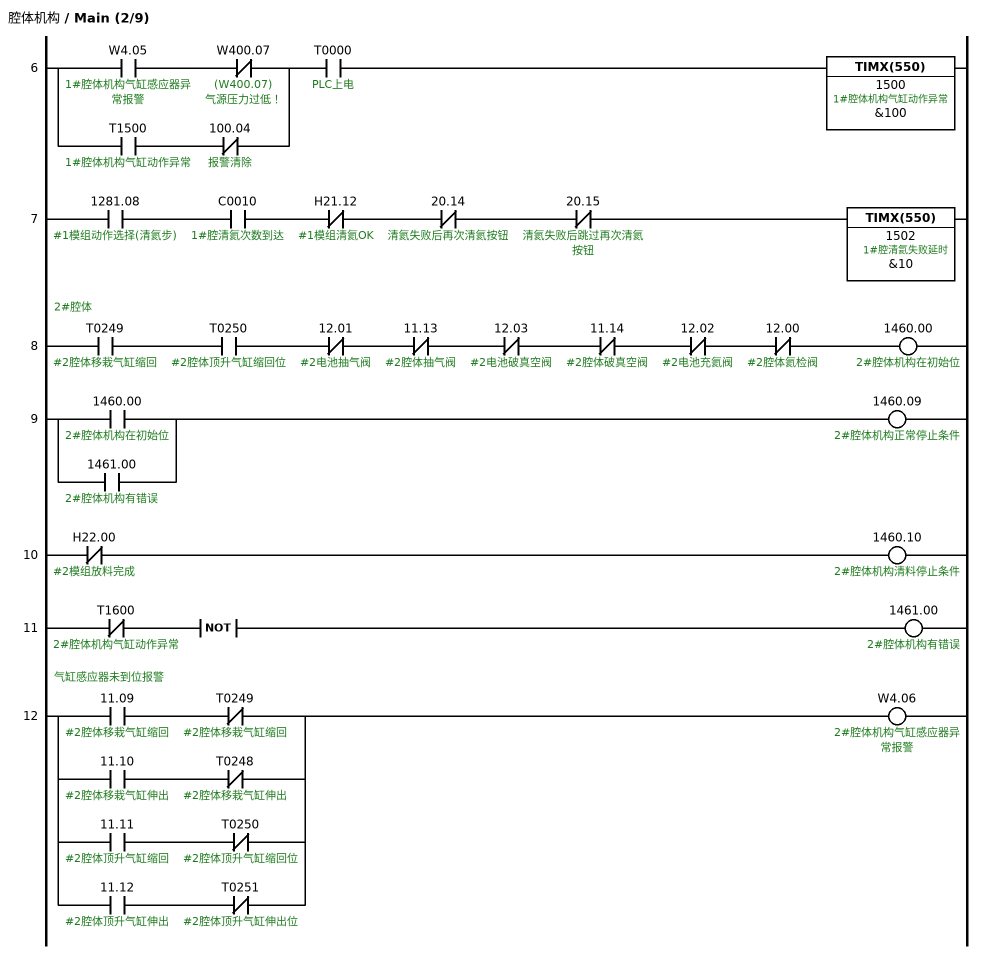
; rung 6
LD W4.05  ; 1#腔体机构气缸感应器异常报警
ANDNOT W400.07  ; (W400.07) 气源压力过低！
LD T1500  ; 1#腔体机构气缸动作异常
ANDNOT 100.04  ; 报警清除
ORLD
AND T0000  ; PLC上电
TIMX(550) 1500 &100  ; 1#腔体机构气缸动作异常
; rung 7
LD 1281.08  ; #1模组动作选择(清氦步)
AND C0010  ; 1#腔清氦次数到达
ANDNOT H21.12  ; #1模组清氦OK
ANDNOT 20.14  ; 清氦失败后再次清氦按钮
ANDNOT 20.15  ; 清氦失败后跳过再次清氦按钮
TIMX(550) 1502 &10  ; 1#腔清氦失败延时
; rung 8: 2#腔体
LD T0249  ; #2腔体移栽气缸缩回
AND T0250  ; #2腔体顶升气缸缩回位
ANDNOT 12.01  ; #2电池抽气阀
ANDNOT 11.13  ; #2腔体抽气阀
ANDNOT 12.03  ; #2电池破真空阀
ANDNOT 11.14  ; #2腔体破真空阀
ANDNOT 12.02  ; #2电池充氦阀
ANDNOT 12.00  ; #2腔体氦检阀
OUT 1460.00  ; 2#腔体机构在初始位
; rung 9
LD 1460.00  ; 2#腔体机构在初始位
OR 1461.00  ; 2#腔体机构有错误
OUT 1460.09  ; 2#腔体机构正常停止条件
; rung 10
LDNOT H22.00  ; #2模组放料完成
OUT 1460.10  ; 2#腔体机构清料停止条件
; rung 11
LDNOT T1600  ; 2#腔体机构气缸动作异常
NOT(520)
OUT 1461.00  ; 2#腔体机构有错误
; rung 12: 气缸感应器未到位报警
LD 11.09  ; #2腔体移栽气缸缩回
ANDNOT T0249  ; #2腔体移栽气缸缩回
LD 11.10  ; #2腔体移栽气缸伸出
ANDNOT T0248  ; #2腔体移栽气缸伸出
ORLD
LD 11.11  ; #2腔体顶升气缸缩回
ANDNOT T0250  ; #2腔体顶升气缸缩回位
ORLD
LD 11.12  ; #2腔体顶升气缸伸出
ANDNOT T0251  ; #2腔体顶升气缸伸出位
ORLD
OUT W4.06  ; 2#腔体机构气缸感应器异常报警

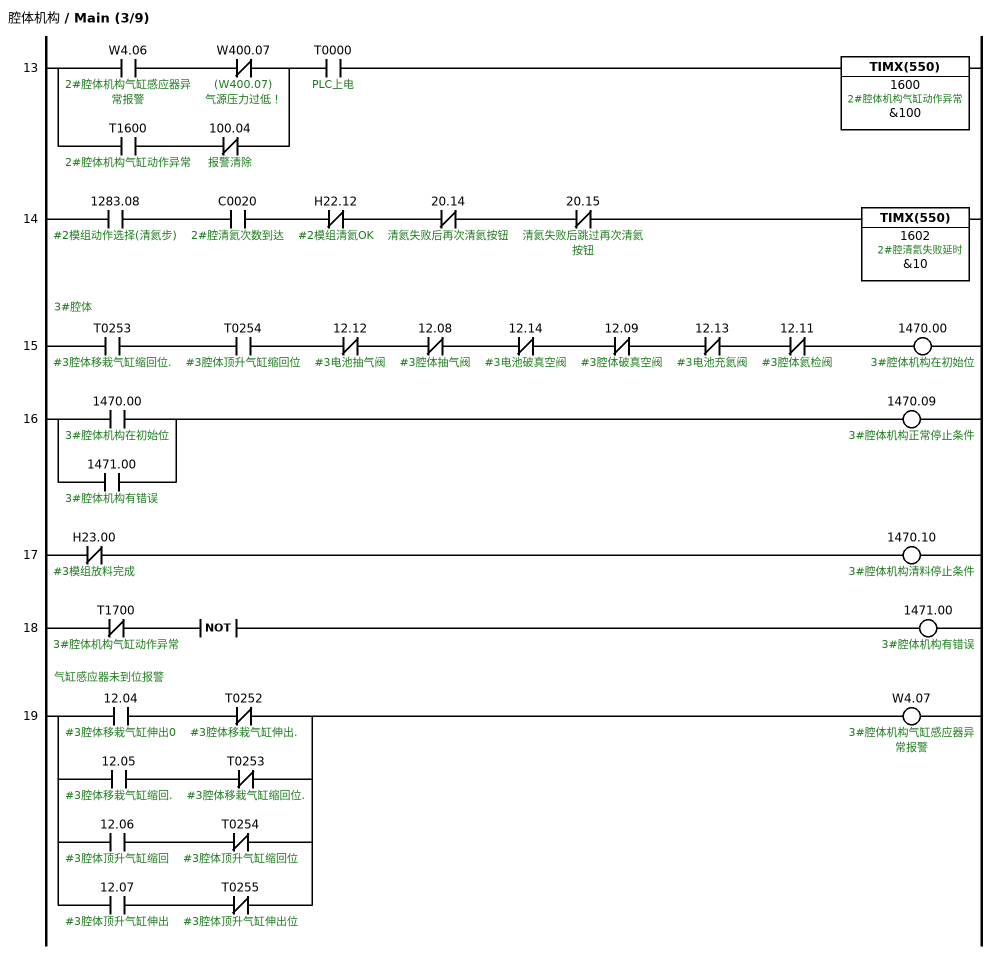
; rung 13
LD W4.06  ; 2#腔体机构气缸感应器异常报警
ANDNOT W400.07  ; (W400.07) 气源压力过低！
LD T1600  ; 2#腔体机构气缸动作异常
ANDNOT 100.04  ; 报警清除
ORLD
AND T0000  ; PLC上电
TIMX(550) 1600 &100  ; 2#腔体机构气缸动作异常
; rung 14
LD 1283.08  ; #2模组动作选择(清氦步)
AND C0020  ; 2#腔清氦次数到达
ANDNOT H22.12  ; #2模组清氦OK
ANDNOT 20.14  ; 清氦失败后再次清氦按钮
ANDNOT 20.15  ; 清氦失败后跳过再次清氦按钮
TIMX(550) 1602 &10  ; 2#腔清氦失败延时
; rung 15: 3#腔体
LD T0253  ; #3腔体移栽气缸缩回位.
AND T0254  ; #3腔体顶升气缸缩回位
ANDNOT 12.12  ; #3电池抽气阀
ANDNOT 12.08  ; #3腔体抽气阀
ANDNOT 12.14  ; #3电池破真空阀
ANDNOT 12.09  ; #3腔体破真空阀
ANDNOT 12.13  ; #3电池充氦阀
ANDNOT 12.11  ; #3腔体氦检阀
OUT 1470.00  ; 3#腔体机构在初始位
; rung 16
LD 1470.00  ; 3#腔体机构在初始位
OR 1471.00  ; 3#腔体机构有错误
OUT 1470.09  ; 3#腔体机构正常停止条件
; rung 17
LDNOT H23.00  ; #3模组放料完成
OUT 1470.10  ; 3#腔体机构清料停止条件
; rung 18
LDNOT T1700  ; 3#腔体机构气缸动作异常
NOT(520)
OUT 1471.00  ; 3#腔体机构有错误
; rung 19: 气缸感应器未到位报警
LD 12.04  ; #3腔体移栽气缸伸出0
ANDNOT T0252  ; #3腔体移栽气缸伸出.
LD 12.05  ; #3腔体移栽气缸缩回.
ANDNOT T0253  ; #3腔体移栽气缸缩回位.
ORLD
LD 12.06  ; #3腔体顶升气缸缩回
ANDNOT T0254  ; #3腔体顶升气缸缩回位
ORLD
LD 12.07  ; #3腔体顶升气缸伸出
ANDNOT T0255  ; #3腔体顶升气缸伸出位
ORLD
OUT W4.07  ; 3#腔体机构气缸感应器异常报警

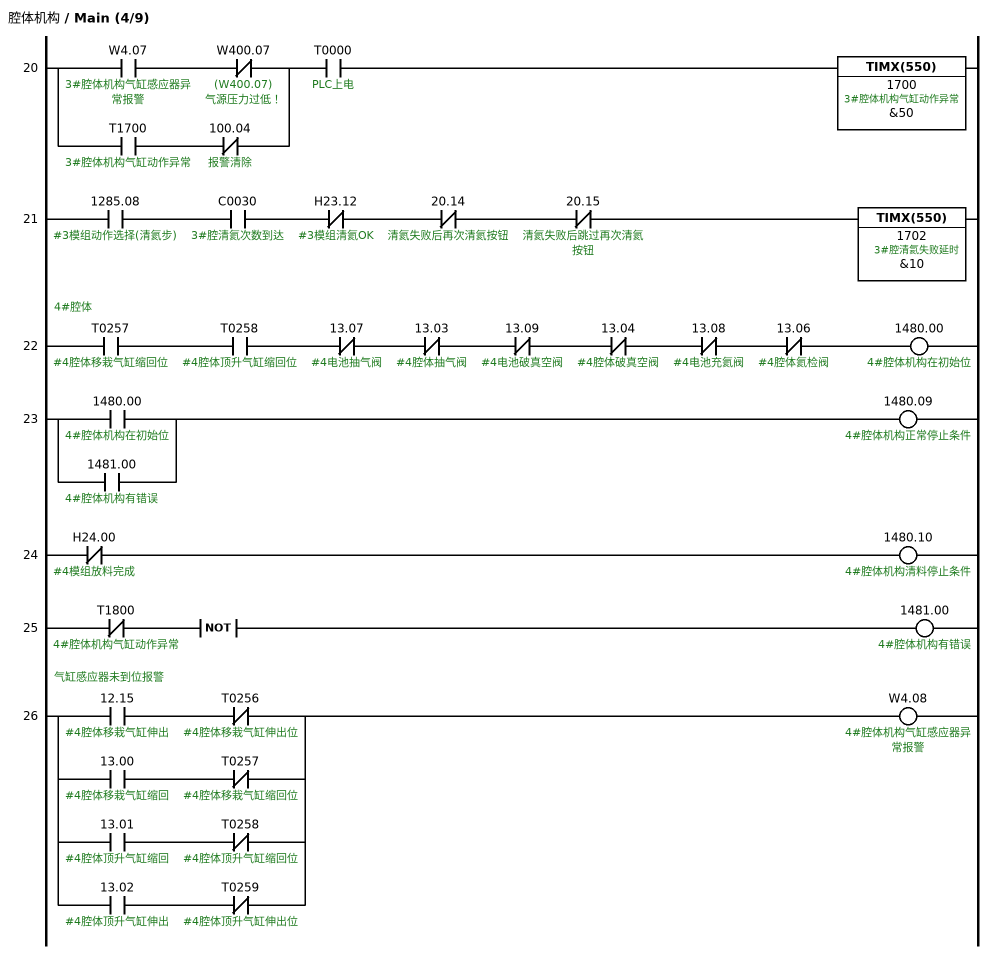
; rung 20
LD W4.07  ; 3#腔体机构气缸感应器异常报警
ANDNOT W400.07  ; (W400.07) 气源压力过低！
LD T1700  ; 3#腔体机构气缸动作异常
ANDNOT 100.04  ; 报警清除
ORLD
AND T0000  ; PLC上电
TIMX(550) 1700 &50  ; 3#腔体机构气缸动作异常
; rung 21
LD 1285.08  ; #3模组动作选择(清氦步)
AND C0030  ; 3#腔清氦次数到达
ANDNOT H23.12  ; #3模组清氦OK
ANDNOT 20.14  ; 清氦失败后再次清氦按钮
ANDNOT 20.15  ; 清氦失败后跳过再次清氦按钮
TIMX(550) 1702 &10  ; 3#腔清氦失败延时
; rung 22: 4#腔体
LD T0257  ; #4腔体移栽气缸缩回位
AND T0258  ; #4腔体顶升气缸缩回位
ANDNOT 13.07  ; #4电池抽气阀
ANDNOT 13.03  ; #4腔体抽气阀
ANDNOT 13.09  ; #4电池破真空阀
ANDNOT 13.04  ; #4腔体破真空阀
ANDNOT 13.08  ; #4电池充氦阀
ANDNOT 13.06  ; #4腔体氦检阀
OUT 1480.00  ; 4#腔体机构在初始位
; rung 23
LD 1480.00  ; 4#腔体机构在初始位
OR 1481.00  ; 4#腔体机构有错误
OUT 1480.09  ; 4#腔体机构正常停止条件
; rung 24
LDNOT H24.00  ; #4模组放料完成
OUT 1480.10  ; 4#腔体机构清料停止条件
; rung 25
LDNOT T1800  ; 4#腔体机构气缸动作异常
NOT(520)
OUT 1481.00  ; 4#腔体机构有错误
; rung 26: 气缸感应器未到位报警
LD 12.15  ; #4腔体移栽气缸伸出
ANDNOT T0256  ; #4腔体移栽气缸伸出位
LD 13.00  ; #4腔体移栽气缸缩回
ANDNOT T0257  ; #4腔体移栽气缸缩回位
ORLD
LD 13.01  ; #4腔体顶升气缸缩回
ANDNOT T0258  ; #4腔体顶升气缸缩回位
ORLD
LD 13.02  ; #4腔体顶升气缸伸出
ANDNOT T0259  ; #4腔体顶升气缸伸出位
ORLD
OUT W4.08  ; 4#腔体机构气缸感应器异常报警

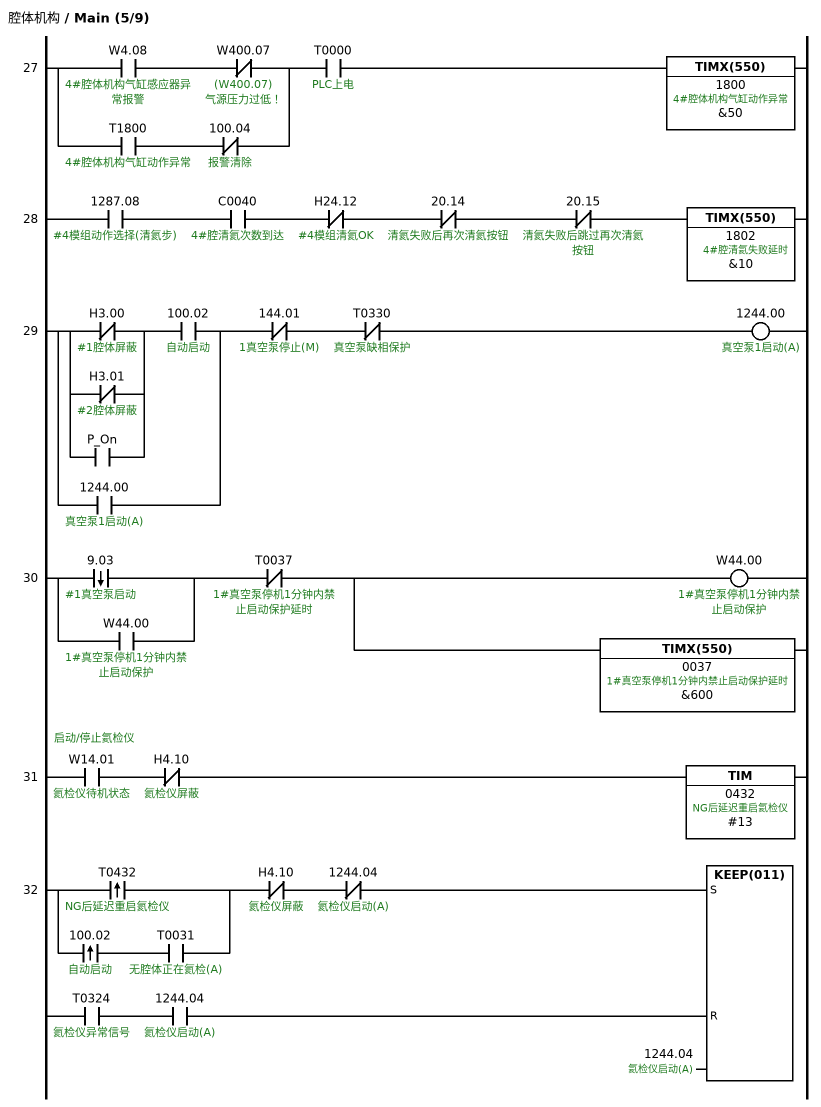
; rung 27
LD W4.08  ; 4#腔体机构气缸感应器异常报警
ANDNOT W400.07  ; (W400.07) 气源压力过低！
LD T1800  ; 4#腔体机构气缸动作异常
ANDNOT 100.04  ; 报警清除
ORLD
AND T0000  ; PLC上电
TIMX(550) 1800 &50  ; 4#腔体机构气缸动作异常
; rung 28
LD 1287.08  ; #4模组动作选择(清氦步)
AND C0040  ; 4#腔清氦次数到达
ANDNOT H24.12  ; #4模组清氦OK
ANDNOT 20.14  ; 清氦失败后再次清氦按钮
ANDNOT 20.15  ; 清氦失败后跳过再次清氦按钮
TIMX(550) 1802 &10  ; 4#腔清氦失败延时
; rung 29
LDNOT H3.00  ; #1腔体屏蔽
ORNOT H3.01  ; #2腔体屏蔽
OR P_On
AND 100.02  ; 自动启动
OR 1244.00  ; 真空泵1启动(A)
ANDNOT 144.01  ; 1真空泵停止(M)
ANDNOT T0330  ; 真空泵缺相保护
OUT 1244.00  ; 真空泵1启动(A)
; rung 30
%LD 9.03  ; #1真空泵启动
OR W44.00  ; 1#真空泵停机1分钟内禁止启动保护
ANDNOT T0037  ; 1#真空泵停机1分钟内禁止启动保护延时
OUT W44.00  ; 1#真空泵停机1分钟内禁止启动保护
TIMX(550) 0037 &600  ; 1#真空泵停机1分钟内禁止启动保护延时
; rung 31: 启动/停止氦检仪
LD W14.01  ; 氦检仪待机状态
ANDNOT H4.10  ; 氦检仪屏蔽
TIM 0432 #13  ; NG后延迟重启氦检仪
; rung 32
@LD T0432  ; NG后延迟重启氦检仪
@LD 100.02  ; 自动启动
AND T0031  ; 无腔体正在氦检(A)
ORLD
ANDNOT H4.10  ; 氦检仪屏蔽
ANDNOT 1244.04  ; 氦检仪启动(A)
LD T0324  ; 氦检仪异常信号
AND 1244.04  ; 氦检仪启动(A)
KEEP(011) 1244.04  ; 氦检仪启动(A)

